Fanuc TP program (LS listing): OP5_LRG_SEQCHNG_AIR_D.LS

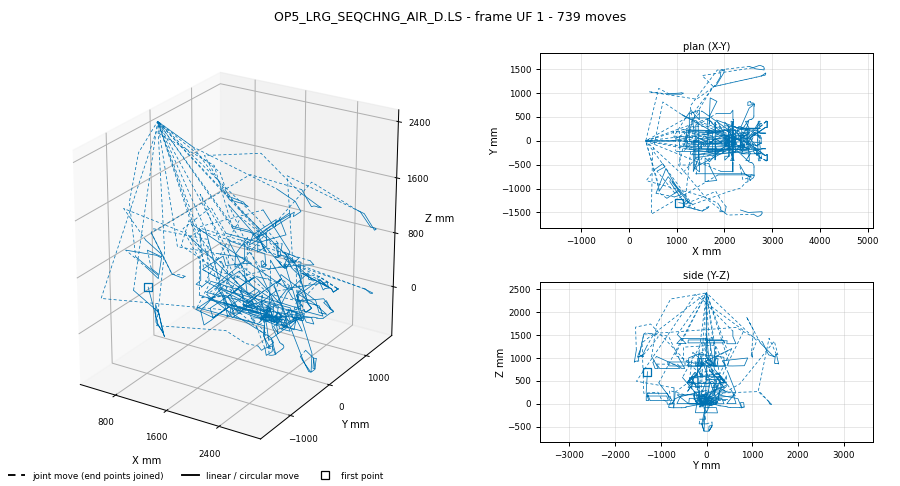
[picture p0: tool path of OP5_LRG_SEQCHNG_AIR_D.LS in frame UF 1, 739 of 740 moves have a stored position in this frame; points joined in program order, loops and branches not executed]
/PROG  OP5_LRG_SEQCHNG_AIR_D
/ATTR
OWNER		= MNEDITOR;
COMMENT		= "Large Main Base";
PROG_SIZE	= 95312;
CREATE		= DATE 26-02-26  TIME 11:37:22;
MODIFIED	= DATE 26-02-26  TIME 13:54:42;
FILE_NAME	= OP5_LRG_;
VERSION		= 0;
LINE_COUNT	= 2634;
MEMORY_SIZE	= 95996;
PROTECT		= READ_WRITE;
TCD:  STACK_SIZE	= 0,
      TASK_PRIORITY	= 50,
      TIME_SLICE	= 0,
      BUSY_LAMP_OFF	= 0,
      ABORT_REQUEST	= 0,
      PAUSE_REQUEST	= 0;
DEFAULT_GROUP	= 1,1,*,*,*;
CONTROL_CODE	= 00000000 00000000;
/APPL
  ARC Welding Equipment : 1,*,*,*,*;

MPAS ;
MPAS_NUM_PASSES        : 0;
MPAS_LAST_PASS         : 0;
MPAS_CURRENT_PASS      : 0;
MPAS_STATUS_PASS       : 0;
/MN
   1:  !********** WAR HAMMER ********** ;
   2:  !*------- FRAME LARGE ----------* ;
   3:  !*-- WELD SEQUENCE CHANGE 2026--* ;
   4:  !*------- FR500 CELL: D --------* ;
   5:  !******************************** ;
   6:   ;
   7:  CALL HOME    ;
   8:  UFRAME_NUM=1 ;
   9:  //DO[17:ON :SCAN ZONE2]=OFF ;
  10:   ;
  11:  !********POSITIONER MOVE******** ;
  12:J P[1] 85% CNT40    ;
  13:   ;
  14:L P[3] 1000mm/sec CNT40    ;
  15:   ;
  16:  !FR50L1000 ;
  17:  IF R[15:TECH HOLD]=1002,CALL TECH_HOLD ;
  18:   ;
  19:  !TO SKIP FRONT BUMPER WELDS ;
  20:  CALL ARC_DISABLE_FRONT_BMPR_LRG(0) ;
  21:   ;
  22:   ;
  23:   ;
  24:L P[5] 1000mm/sec FINE
    :  Arc Start[6]    ;
  25:  Weave Sine[6] ;
  26:  Track TAST[6] ;
  27:L P[6] WELD_SPEED FINE
    :  Arc End[6]    ;
  28:  Weave End ;
  29:  Track End ;
  30:   ;
  31:   ;
  32:   ;
  33:   ;
  34:L P[8] 800mm/sec CNT30    ;
  35:   ;
  36:L P[9] 1000mm/sec CNT30    ;
  37:   ;
  38:   ;
  39:  !FR50L1001 ;
  40:  IF R[15:TECH HOLD]=1003,CALL TECH_HOLD ;
  41:   ;
  42:   ;
  43:   ;
  44:   ;
  45:L P[10] 1000mm/sec FINE
    :  Arc Start[6]    ;
  46:  Weave Sine[6] ;
  47:  Track TAST[6] ;
  48:L P[11] WELD_SPEED FINE
    :  Arc End[6]    ;
  49:  Weave End ;
  50:  Track End ;
  51:   ;
  52:   ;
  53:   ;
  54:L P[12] 1000mm/sec CNT100    ;
  55:   ;
  56:   ;
  57:  !FR50L1002 ;
  58:  IF R[15:TECH HOLD]=1004,CALL TECH_HOLD ;
  59:   ;
  60:   ;
  61:L P[13] 1000mm/sec CNT70    ;
  62:   ;
  63:   ;
  64:   ;
  65:L P[14] 1000mm/sec FINE
    :  Arc Start[6]    ;
  66:  Weave Sine[6] ;
  67:  Track TAST[6] ;
  68:L P[15] WELD_SPEED FINE
    :  Arc End[6]    ;
  69:  Weave End ;
  70:  Track End ;
  71:   ;
  72:   ;
  73:   ;
  74:  CALL ARC_DISABLE_FRONT_BMPR_LRG(1) ;
  75:   ;
  76:L P[16] 1000mm/sec CNT100    ;
  77:   ;
  78:  !HOME ;
  79:J P[4] 70% CNT30    ;
  80:   ;
  81:  !********POSITIONER MOVE******** ;
  82:J P[17] 85% CNT30    ;
  83:   ;
  84:J P[18] 50% CNT100    ;
  85:   ;
  86:L P[19] 1000mm/sec CNT100    ;
  87:   ;
  88:   ;
  89:  !FR50L1003 ;
  90:  IF R[15:TECH HOLD]=1005,CALL TECH_HOLD ;
  91:   ;
  92:   ;
  93:L P[20] 1000mm/sec CNT25    ;
  94:   ;
  95:   ;
  96:   ;
  97:L P[21] 1000mm/sec FINE
    :  Arc Start[6]    ;
  98:  Weave Sine[6] ;
  99:  Track TAST[6] ;
 100:L P[22] WELD_SPEED CNT100    ;
 101:L P[23] WELD_SPEED FINE
    :  Arc End[6]    ;
 102:  Track End ;
 103:  Weave End ;
 104:   ;
 105:   ;
 106:   ;
 107:L P[24] 1000mm/sec CNT30    ;
 108:   ;
 109:   ;
 110:  !FR50L1010 ;
 111:  IF R[15:TECH HOLD]=1012,CALL TECH_HOLD ;
 112:   ;
 113:   ;
 114:L P[25] 1000mm/sec CNT30    ;
 115:   ;
 116:   ;
 117:   ;
 118:L P[26] 1000mm/sec FINE
    :  Arc Start[6]    ;
 119:  Weave Sine[6] ;
 120:  Track TAST[6] ;
 121:L P[27] WELD_SPEED CNT100    ;
 122:L P[28] WELD_SPEED FINE
    :  Arc End[6]    ;
 123:  Weave End ;
 124:  Track End ;
 125:   ;
 126:   ;
 127:   ;
 128:L P[29] 1000mm/sec CNT25    ;
 129:   ;
 130:   ;
 131:  !FR50L1020 ;
 132:  IF R[15:TECH HOLD]=1022,CALL TECH_HOLD ;
 133:   ;
 134:   ;
 135:J P[30] 50% CNT25    ;
 136:   ;
 137:   ;
 138:   ;
 139:L P[31] 1000mm/sec FINE
    :  Arc Start[6]    ;
 140:  Weave Sine[6] ;
 141:  Track TAST[6] ;
 142:L P[32] WELD_SPEED FINE
    :  Arc End[6]    ;
 143:  Weave End ;
 144:  Track End ;
 145:   ;
 146:   ;
 147:   ;
 148:L P[33] 1000mm/sec CNT30    ;
 149:   ;
 150:L P[34] 1000mm/sec CNT30    ;
 151:   ;
 152:   ;
 153:  !FR50L1030 ;
 154:  IF R[15:TECH HOLD]=1032,CALL TECH_HOLD ;
 155:   ;
 156:   ;
 157:   ;
 158:   ;
 159:L P[35] 1000mm/sec FINE
    :  Arc Start[6]    ;
 160:  Weave Sine[6] ;
 161:  Track TAST[6] ;
 162:L P[36] WELD_SPEED FINE
    :  Arc End[6]    ;
 163:  Weave End ;
 164:  Track End ;
 165:   ;
 166:   ;
 167:   ;
 168:L P[37] 1000mm/sec CNT50    ;
 169:   ;
 170:J P[38] 50% CNT50    ;
 171:   ;
 172:L P[39] 1000mm/sec CNT25    ;
 173:   ;
 174:   ;
 175:  !FR50L1040 ;
 176:  IF R[15:TECH HOLD]=1042,CALL TECH_HOLD ;
 177:   ;
 178:   ;
 179:   ;
 180:   ;
 181:L P[40] 1000mm/sec FINE
    :  Arc Start[6]    ;
 182:  Weave Sine[6] ;
 183:L P[41] WELD_SPEED FINE
    :  Arc End[6]    ;
 184:  Weave End ;
 185:   ;
 186:   ;
 187:   ;
 188:L P[42] 1000mm/sec CNT30    ;
 189:   ;
 190:L P[43] 1000mm/sec CNT70    ;
 191:   ;
 192:J P[44] 50% CNT50    ;
 193:   ;
 194:L P[45] 1000mm/sec CNT30    ;
 195:   ;
 196:   ;
 197:  !FR50L1050 ;
 198:  IF R[15:TECH HOLD]=1052,CALL TECH_HOLD ;
 199:   ;
 200:   ;
 201:   ;
 202:   ;
 203:L P[46] 1000mm/sec FINE
    :  Arc Start[6]    ;
 204:  Weave Sine[6] ;
 205:L P[47] WELD_SPEED FINE
    :  Arc End[6]    ;
 206:  Weave End ;
 207:   ;
 208:   ;
 209:   ;
 210:L P[48] 1000mm/sec CNT80    ;
 211:   ;
 212:J P[49] 50% CNT25    ;
 213:   ;
 214:L P[50] 1000mm/sec CNT25    ;
 215:   ;
 216:   ;
 217:  !FR50L1060 ;
 218:  IF R[15:TECH HOLD]=1062,CALL TECH_HOLD ;
 219:   ;
 220:   ;
 221:   ;
 222:   ;
 223:L P[51] 1000mm/sec FINE
    :  Arc Start[6]    ;
 224:  Weave Sine[6] ;
 225:L P[52] WELD_SPEED FINE
    :  Arc End[6]    ;
 226:  Weave End ;
 227:   ;
 228:   ;
 229:   ;
 230:L P[53] 500mm/sec CNT100    ;
 231:   ;
 232:L P[54] 1500mm/sec CNT35    ;
 233:   ;
 234:J P[55] 50% CNT30    ;
 235:   ;
 236:L P[56] 1000mm/sec CNT30    ;
 237:   ;
 238:   ;
 239:  !FR50L1070 ;
 240:  IF R[15:TECH HOLD]=1072,CALL TECH_HOLD ;
 241:   ;
 242:   ;
 243:   ;
 244:   ;
 245:L P[57] 1000mm/sec FINE
    :  Arc Start[6]    ;
 246:  Weave Sine[6] ;
 247:  Track TAST[6] ;
 248:L P[58] WELD_SPEED FINE
    :  Arc End[6]    ;
 249:  Weave End ;
 250:  Track End ;
 251:   ;
 252:   ;
 253:   ;
 254:L P[59] 1000mm/sec CNT100    ;
 255:   ;
 256:L P[60] 1000mm/sec CNT80    ;
 257:   ;
 258:   ;
 259:  !FR50L1080 ;
 260:  IF R[15:TECH HOLD]=1082,CALL TECH_HOLD ;
 261:   ;
 262:   ;
 263:   ;
 264:   ;
 265:L P[61] 1000mm/sec FINE
    :  Arc Start[6]    ;
 266:  Weave Sine[6] ;
 267:  Track TAST[6] ;
 268:L P[62] WELD_SPEED FINE
    :  Arc End[6]    ;
 269:  Weave End ;
 270:  Track End ;
 271:   ;
 272:   ;
 273:   ;
 274:J P[63] 30% CNT100    ;
 275:   ;
 276:J P[64] 50% CNT100    ;
 277:   ;
 278:L P[65] 1000mm/sec CNT80    ;
 279:   ;
 280:   ;
 281:  !FR50L1090 ;
 282:  IF R[15:TECH HOLD]=1092,CALL TECH_HOLD ;
 283:  !10MM PASS ;
 284:   ;
 285:   ;
 286:   ;
 287:   ;
 288:L P[66] 1000mm/sec FINE
    :  Arc Start[6]    ;
 289:  Weave Sine[6] ;
 290:  Track TAST[6] RPM[1] ;
 291:L P[67] WELD_SPEED CNT100    ;
 292:L P[68] WELD_SPEED CNT100    ;
 293:C P[69]
    :  P[70] WELD_SPEED CNT100    ;
 294:L P[71] WELD_SPEED FINE
    :  Arc End[6]    ;
 295:  Track End ;
 296:  Weave End ;
 297:   ;
 298:   ;
 299:   ;
 300:J P[72] 16% CNT25    ;
 301:   ;
 302:J P[74] 50% CNT25    ;
 303:   ;
 304:L P[75] 1000mm/sec CNT25    ;
 305:   ;
 306:   ;
 307:  !FR50L1100 ;
 308:  IF R[15:TECH HOLD]=1102,CALL TECH_HOLD ;
 309:   ;
 310:   ;
 311:   ;
 312:   ;
 313:L P[76] 1000mm/sec FINE
    :  Arc Start[6]    ;
 314:  Weave Sine[6] ;
 315:  Track TAST[6] RPM[2] ;
 316:L P[77] WELD_SPEED CNT100    ;
 317:L P[78] WELD_SPEED CNT100    ;
 318:C P[79]
    :  P[80] WELD_SPEED CNT100    ;
 319:L P[81] WELD_SPEED FINE
    :  Arc End[6]    ;
 320:  Weave End ;
 321:  Track End ;
 322:   ;
 323:   ;
 324:   ;
 325:J P[82] 50% CNT10    ;
 326:   ;
 327:J P[83] 50% CNT80    ;
 328:   ;
 329:L P[84] 1000mm/sec CNT25    ;
 330:   ;
 331:   ;
 332:  !FR50L1110MP1 ;
 333:  IF R[15:TECH HOLD]=1112,CALL TECH_HOLD ;
 334:   ;
 335:   ;
 336:  MP Offset  PR[3] RPM[1] ;
 337:   ;
 338:   ;
 339:L P[66] 1000mm/sec FINE
    :  Arc Start[6]    ;
 340:  Weave Sine[6] ;
 341:L P[67] WELD_SPEED CNT100    ;
 342:L P[68] WELD_SPEED CNT100    ;
 343:C P[69]
    :  P[70] WELD_SPEED CNT100    ;
 344:L P[71] WELD_SPEED FINE
    :  Arc End[6]    ;
 345:  Track End ;
 346:  Weave End ;
 347:   ;
 348:   ;
 349:  MP Offset End ;
 350:   ;
 351:J P[91] 40% CNT10    ;
 352:   ;
 353:J P[92] 50% CNT30    ;
 354:   ;
 355:L P[93] 1000mm/sec CNT25    ;
 356:   ;
 357:   ;
 358:  !FR50M1110MP2 ;
 359:   ;
 360:   ;
 361:  MP Offset  PR[4] RPM[1] ;
 362:   ;
 363:   ;
 364:L P[66] 1000mm/sec FINE
    :  Arc Start[6]    ;
 365:  Weave Sine[6] ;
 366:L P[67] WELD_SPEED CNT100    ;
 367:L P[68] WELD_SPEED CNT100    ;
 368:C P[69]
    :  P[70] WELD_SPEED CNT100    ;
 369:L P[71] WELD_SPEED FINE
    :  Arc End[6]    ;
 370:  Track End ;
 371:  Weave End ;
 372:   ;
 373:  MP Offset End ;
 374:   ;
 375:J P[100] 50% CNT25    ;
 376:   ;
 377:J P[102] 50% CNT25    ;
 378:   ;
 379:L P[103] 1000mm/sec CNT25    ;
 380:   ;
 381:   ;
 382:  !FR50L1120MP3 ;
 383:  IF R[15:TECH HOLD]=1122,CALL TECH_HOLD ;
 384:   ;
 385:   ;
 386:  MP Offset  PR[1] RPM[2] ;
 387:   ;
 388:   ;
 389:L P[76] 1000mm/sec FINE
    :  Arc Start[6]    ;
 390:  Weave Sine[6] ;
 391:L P[77] WELD_SPEED CNT100    ;
 392:L P[78] WELD_SPEED CNT100    ;
 393:C P[79]
    :  P[80] WELD_SPEED CNT100    ;
 394:L P[81] WELD_SPEED FINE
    :  Arc End[6]    ;
 395:  Weave End ;
 396:  Track End ;
 397:   ;
 398:   ;
 399:  MP Offset End ;
 400:   ;
 401:J P[110] 50% CNT25    ;
 402:   ;
 403:J P[111] 50% CNT25    ;
 404:   ;
 405:L P[112] 1000mm/sec CNT25    ;
 406:   ;
 407:   ;
 408:  !FR501130MP4 ;
 409:   ;
 410:   ;
 411:  MP Offset  PR[2] RPM[2] ;
 412:   ;
 413:L P[76] 1000mm/sec FINE
    :  Arc Start[6]    ;
 414:  Weave Sine[6] ;
 415:L P[77] WELD_SPEED CNT100    ;
 416:L P[78] WELD_SPEED CNT100    ;
 417:C P[79]
    :  P[80] WELD_SPEED CNT100    ;
 418:L P[81] WELD_SPEED FINE
    :  Arc End[6]    ;
 419:  Weave End ;
 420:  Track End ;
 421:   ;
 422:  MP Offset End ;
 423:   ;
 424:J P[119] 50% CNT25    ;
 425:   ;
 426:J P[121] 50% CNT25    ;
 427:   ;
 428:L P[122] 1000mm/sec CNT25    ;
 429:   ;
 430:   ;
 431:  !FR50L1140 ;
 432:  IF R[15:TECH HOLD]=1142,CALL TECH_HOLD ;
 433:   ;
 434:   ;
 435:   ;
 436:   ;
 437:L P[185] 1000mm/sec FINE
    :  Arc Start[8]    ;
 438:  Weave Sine[8] ;
 439:L P[186] WELD_SPEED CNT100    ;
 440:C P[187]
    :  P[188] WELD_SPEED FINE
    :  Arc End[8]    ;
 441:  Weave End ;
 442:   ;
 443:   ;
 444:   ;
 445:L P[127] 1000mm/sec CNT25    ;
 446:   ;
 447:J P[128] 50% CNT25    ;
 448:   ;
 449:   ;
 450:  !FR50L1141 ;
 451:  IF R[15:TECH HOLD]=1143,CALL TECH_HOLD ;
 452:   ;
 453:   ;
 454:   ;
 455:   ;
 456:L P[192] 1000mm/sec FINE
    :  Arc Start[8]    ;
 457:  Weave Sine[8] ;
 458:L P[193] WELD_SPEED CNT100    ;
 459:C P[194]
    :  P[197] WELD_SPEED FINE
    :  Arc End[8]    ;
 460:  Weave End ;
 461:   ;
 462:   ;
 463:   ;
 464:L P[133] 1000mm/sec CNT25    ;
 465:   ;
 466:L P[134] 1000mm/sec CNT25    ;
 467:   ;
 468:J P[135] 50% CNT25    ;
 469:   ;
 470:L P[136] 1000mm/sec CNT50    ;
 471:   ;
 472:   ;
 473:  !FR50L1150 ;
 474:  IF R[15:TECH HOLD]=1152,CALL TECH_HOLD ;
 475:   ;
 476:   ;
 477:   ;
 478:   ;
 479:L P[198] 1000mm/sec FINE
    :  Arc Start[6]    ;
 480:  Weave Sine[6] ;
 481:  Track TAST[6] ;
 482:L P[199] WELD_SPEED FINE
    :  Arc End[6]    ;
 483:  Weave End ;
 484:  Track End ;
 485:   ;
 486:   ;
 487:   ;
 488:L P[139] 1000mm/sec CNT100    ;
 489:   ;
 490:L P[140] 1000mm/sec CNT50    ;
 491:   ;
 492:   ;
 493:  !FR50L1160 ;
 494:  IF R[15:TECH HOLD]=1162,CALL TECH_HOLD ;
 495:   ;
 496:   ;
 497:   ;
 498:L P[203] 1000mm/sec FINE
    :  Arc Start[6]    ;
 499:  Weave Sine[6] ;
 500:  Track TAST[6] ;
 501:L P[204] WELD_SPEED FINE
    :  Arc End[6]    ;
 502:  Weave End ;
 503:  Track End ;
 504:   ;
 505:   ;
 506:   ;
 507:L P[143] 1000mm/sec CNT30    ;
 508:   ;
 509:  !********POSITIONER MOVE******** ;
 510:J P[144] 85% CNT30    ;
 511:   ;
 512:L P[145] 1000mm/sec CNT100    ;
 513:   ;
 514:   ;
 515:  !FR50L1170 ;
 516:  IF R[15:TECH HOLD]=1172,CALL TECH_HOLD ;
 517:   ;
 518:   ;
 519:   ;
 520:   ;
 521:L P[205] 1000mm/sec FINE
    :  Arc Start[6]    ;
 522:  Weave Sine[6] ;
 523:  Track TAST[6] ;
 524:L P[208] WELD_SPEED FINE
    :  Arc End[6]    ;
 525:  Weave End ;
 526:  Track End ;
 527:   ;
 528:   ;
 529:   ;
 530:L P[148] 1000mm/sec CNT100    ;
 531:   ;
 532:L P[149] 1500mm/sec CNT100    ;
 533:   ;
 534:   ;
 535:  !FR50L1180 ;
 536:  IF R[15:TECH HOLD]=1182,CALL TECH_HOLD ;
 537:   ;
 538:   ;
 539:   ;
 540:   ;
 541:L P[209] 1000mm/sec FINE
    :  Arc Start[6]    ;
 542:  Weave Sine[6] ;
 543:  Track TAST[6] ;
 544:L P[212] WELD_SPEED FINE
    :  Arc End[6]    ;
 545:  Weave End ;
 546:  Track End ;
 547:   ;
 548:   ;
 549:   ;
 550:L P[152] 1000mm/sec CNT100    ;
 551:   ;
 552:  !HOME ;
 553:J P[7] 100% CNT30    ;
 554:   ;
 555:  !********POSITIONER MOVE******** ;
 556:J P[153] 80% CNT30    ;
 557:   ;
 558:J P[154] 50% CNT100    ;
 559:   ;
 560:L P[155] 1000mm/sec CNT25    ;
 561:   ;
 562:   ;
 563:  !FR50L1210 ;
 564:  IF R[15:TECH HOLD]=1212,CALL TECH_HOLD ;
 565:   ;
 566:   ;
 567:   ;
 568:   ;
 569:L P[213] 1000mm/sec FINE
    :  Arc Start[6]    ;
 570:  Weave Sine[6] ;
 571:  Track TAST[6] ;
 572:L P[216] WELD_SPEED CNT100    ;
 573:L P[217] WELD_SPEED FINE
    :  Arc End[6]    ;
 574:  Weave End ;
 575:  Track End ;
 576:   ;
 577:   ;
 578:   ;
 579:L P[159] 1000mm/sec CNT25    ;
 580:   ;
 581:L P[160] 1000mm/sec CNT25    ;
 582:   ;
 583:   ;
 584:  !FR50L1220 ;
 585:  IF R[15:TECH HOLD]=1222,CALL TECH_HOLD ;
 586:   ;
 587:   ;
 588:   ;
 589:   ;
 590:L P[218] 1000mm/sec FINE
    :  Arc Start[6]    ;
 591:  Weave Sine[6] ;
 592:  Track TAST[6] ;
 593:L P[221] WELD_SPEED CNT100    ;
 594:L P[222] WELD_SPEED FINE
    :  Arc End[6]    ;
 595:  Weave End ;
 596:  Track End ;
 597:   ;
 598:   ;
 599:   ;
 600:L P[163] 1000mm/sec CNT80    ;
 601:   ;
 602:L P[164] 1200mm/sec CNT25    ;
 603:   ;
 604:   ;
 605:  !FR50L1230 ;
 606:  IF R[15:TECH HOLD]=1232,CALL TECH_HOLD ;
 607:   ;
 608:   ;
 609:   ;
 610:   ;
 611:L P[223] 1000mm/sec FINE
    :  Arc Start[6]    ;
 612:  Weave Sine[6] ;
 613:  Track TAST[6] ;
 614:L P[226] WELD_SPEED CNT100    ;
 615:L P[227] WELD_SPEED FINE
    :  Arc End[6]    ;
 616:  Weave End ;
 617:  Track End ;
 618:   ;
 619:   ;
 620:   ;
 621:L P[167] 1000mm/sec CNT25    ;
 622:   ;
 623:L P[168] 1000mm/sec CNT25    ;
 624:   ;
 625:   ;
 626:  !FR50L1240 ;
 627:  IF R[15:TECH HOLD]=1242,CALL TECH_HOLD ;
 628:   ;
 629:   ;
 630:   ;
 631:   ;
 632:L P[228] 1000mm/sec FINE
    :  Arc Start[6]    ;
 633:  Weave Sine[6] ;
 634:  Track TAST[6] ;
 635:L P[229] WELD_SPEED CNT100    ;
 636:L P[231] WELD_SPEED FINE
    :  Arc End[6]    ;
 637:  Weave End ;
 638:  Track End ;
 639:   ;
 640:   ;
 641:   ;
 642:L P[172] 1000mm/sec CNT25    ;
 643:   ;
 644:L P[173] 1000mm/sec CNT100    ;
 645:   ;
 646:  !HOME ;
 647:J P[116] 100% CNT100    ;
 648:   ;
 649:   ;
 650:  !********POSITIONER MOVE******** ;
 651:J P[174] 85% FINE    ;
 652:   ;
 653:  CALL T_CLEAN    ;
 654:   ;
 655:J P[175] 50% CNT35    ;
 656:   ;
 657:L P[176] 1000mm/sec CNT25    ;
 658:   ;
 659:   ;
 660:  !FR50L1250 ;
 661:  IF R[15:TECH HOLD]=1252,CALL TECH_HOLD ;
 662:   ;
 663:   ;
 664:   ;
 665:   ;
 666:L P[232] 1000mm/sec FINE
    :  Arc Start[6]    ;
 667:  Weave Sine[6] ;
 668:  Track TAST[6] ;
 669:L P[236] WELD_SPEED CNT100    ;
 670:L P[237] WELD_SPEED CNT100    ;
 671:L P[238] WELD_SPEED FINE
    :  Arc End[6]    ;
 672:  Weave End ;
 673:  Track End ;
 674:   ;
 675:   ;
 676:   ;
 677:L P[181] 1000mm/sec CNT100    ;
 678:   ;
 679:J P[182] 50% CNT100    ;
 680:   ;
 681:L P[184] 500mm/sec CNT100    ;
 682:   ;
 683:   ;
 684:  !FR50L1260 ;
 685:  IF R[15:TECH HOLD]=1262,CALL TECH_HOLD ;
 686:   ;
 687:   ;
 688:   ;
 689:   ;
 690:L P[239] 1000mm/sec FINE
    :  Arc Start[6]    ;
 691:  Weave Sine[6] ;
 692:  Track TAST[6] ;
 693:L P[244] WELD_SPEED CNT100    ;
 694:L P[245] WELD_SPEED CNT100    ;
 695:L P[246] WELD_SPEED FINE
    :  Arc End[6]    ;
 696:  Weave End ;
 697:  Track End ;
 698:   ;
 699:   ;
 700:   ;
 701:L P[189] 1000mm/sec CNT25    ;
 702:   ;
 703:J P[190] 50% CNT25    ;
 704:   ;
 705:L P[191] 1000mm/sec CNT25    ;
 706:   ;
 707:   ;
 708:  !FR50L1270 ;
 709:  IF R[15:TECH HOLD]=1272,CALL TECH_HOLD ;
 710:   ;
 711:   ;
 712:   ;
 713:   ;
 714:L P[247] 1000mm/sec FINE
    :  Arc Start[6]    ;
 715:  Weave Sine[6] ;
 716:  Track TAST[6] ;
 717:L P[250] WELD_SPEED CNT100    ;
 718:  Track End ;
 719:L P[251] WELD_SPEED FINE
    :  Arc End[6]    ;
 720:  Weave End ;
 721:  Track End ;
 722:   ;
 723:   ;
 724:   ;
 725:L P[195] 1000mm/sec CNT80    ;
 726:   ;
 727:L P[196] 1000mm/sec CNT100    ;
 728:   ;
 729:   ;
 730:  !FR50L1280 ;
 731:  IF R[15:TECH HOLD]=1282,CALL TECH_HOLD ;
 732:   ;
 733:   ;
 734:   ;
 735:   ;
 736:L P[253] 1000mm/sec FINE
    :  Arc Start[6]    ;
 737:  Weave Sine[6] ;
 738:  Track TAST[6] ;
 739:L P[254] WELD_SPEED CNT100    ;
 740:  Track End ;
 741:L P[255] WELD_SPEED FINE
    :  Arc End[6]    ;
 742:  Weave End ;
 743:  Track End ;
 744:   ;
 745:   ;
 746:   ;
 747:L P[200] 1000mm/sec CNT25    ;
 748:   ;
 749:J P[201] 50% CNT25    ;
 750:   ;
 751:L P[202] 1000mm/sec CNT25    ;
 752:   ;
 753:   ;
 754:  !FR50L1290 ;
 755:  IF R[15:TECH HOLD]=1292,CALL TECH_HOLD ;
 756:   ;
 757:   ;
 758:   ;
 759:   ;
 760:L P[257] 1000mm/sec FINE
    :  Arc Start[6]    ;
 761:  Weave Sine[6] ;
 762:  Track TAST[6] ;
 763:L P[258] WELD_SPEED CNT100    ;
 764:L P[259] WELD_SPEED FINE
    :  Arc End[6]    ;
 765:  Weave End ;
 766:  Track End ;
 767:L P[262] 1000mm/sec FINE
    :  Arc Start[6]    ;
 768:  Weave Sine[6] ;
 769:  Track TAST[6] ;
 770:L P[263] WELD_SPEED CNT100    ;
 771:L P[264] WELD_SPEED FINE
    :  Arc End[6]    ;
 772:  Weave End ;
 773:  Track End ;
 774:   ;
 775:   ;
 776:   ;
 777:L P[206] 1000mm/sec CNT100    ;
 778:   ;
 779:L P[207] 1000mm/sec CNT100    ;
 780:   ;
 781:   ;
 782:  !FR50L1300 ;
 783:  IF R[15:TECH HOLD]=1302,CALL TECH_HOLD ;
 784:   ;
 785:   ;
 786:   ;
 787:L P[90] 1000mm/sec FINE
    :  Arc Start[6]    ;
 788:  Weave Sine[6] ;
 789:  Track TAST[6] ;
 790:L P[98] WELD_SPEED CNT100    ;
 791:L P[101] WELD_SPEED FINE
    :  Arc End[6]    ;
 792:  Weave End ;
 793:  Track End ;
 794:   ;
 795:   ;
 796:L P[210] 1000mm/sec CNT100    ;
 797:   ;
 798:L P[211] 1000mm/sec CNT100    ;
 799:   ;
 800:   ;
 801:  !FR50L1310 ;
 802:  IF R[15:TECH HOLD]=1312,CALL TECH_HOLD ;
 803:   ;
 804:   ;
 805:   ;
 806:   ;
 807:L P[266] 1000mm/sec FINE
    :  Arc Start[6]    ;
 808:  Weave Sine[6] ;
 809:  Track TAST[6] ;
 810:L P[267] WELD_SPEED FINE
    :  Arc End[6]    ;
 811:  Weave End ;
 812:  Track End ;
 813:   ;
 814:   ;
 815:   ;
 816:L P[214] 1000mm/sec CNT100    ;
 817:   ;
 818:L P[215] 1000mm/sec CNT100    ;
 819:   ;
 820:   ;
 821:  !FR50L1320 ;
 822:  IF R[15:TECH HOLD]=1322,CALL TECH_HOLD ;
 823:   ;
 824:   ;
 825:   ;
 826:   ;
 827:L P[268] 1000mm/sec FINE
    :  Arc Start[6]    ;
 828:  Weave Sine[6] ;
 829:  Track TAST[6] ;
 830:L P[274] WELD_SPEED CNT100    ;
 831:L P[275] WELD_SPEED FINE
    :  Arc End[6]    ;
 832:  Weave End ;
 833:  Track End ;
 834:   ;
 835:   ;
 836:   ;
 837:L P[219] 1000mm/sec CNT100    ;
 838:   ;
 839:L P[220] 1000mm/sec CNT100    ;
 840:   ;
 841:J P[73] 50% CNT30    ;
 842:   ;
 843:  !********POSITIONER MOVE******** ;
 844:J P[86] 100% CNT30    ;
 845:   ;
 846:  !FR50L1330 ;
 847:  IF R[15:TECH HOLD]=1332,CALL TECH_HOLD ;
 848:   ;
 849:   ;
 850:J P[327] 40% CNT10    ;
 851:   ;
 852:   ;
 853:   ;
 854:L P[277] 1000mm/sec FINE
    :  Arc Start[8]    ;
 855:  Weave Sine[8] ;
 856:L P[278] WELD_SPEED FINE
    :  Arc End[8]    ;
 857:  Weave End ;
 858:   ;
 859:   ;
 860:   ;
 861:J P[85] 50% CNT30    ;
 862:   ;
 863:L P[233] 1000mm/sec CNT25    ;
 864:   ;
 865:  !********POSITIONER MOVE******** ;
 866:J P[225] 80% CNT20    ;
 867:   ;
 868:   ;
 869:   ;
 870:  !FR50L1340 ;
 871:  IF R[15:TECH HOLD]=1342,CALL TECH_HOLD ;
 872:   ;
 873:   ;
 874:   ;
 875:   ;
 876:L P[279] 1000mm/sec FINE
    :  Arc Start[6]    ;
 877:  Weave Sine[6] ;
 878:L P[282] WELD_SPEED FINE
    :  Arc End[6]    ;
 879:  Weave End ;
 880:   ;
 881:   ;
 882:   ;
 883:   ;
 884:  !FR50L1350 ;
 885:  IF R[15:TECH HOLD]=1352,CALL TECH_HOLD ;
 886:   ;
 887:   ;
 888:   ;
 889:   ;
 890:L P[283] 1000mm/sec FINE
    :  Arc Start[6]    ;
 891:  Weave Sine[6] ;
 892:L P[284] WELD_SPEED FINE
    :  Arc End[6]    ;
 893:  Weave End ;
 894:   ;
 895:   ;
 896:   ;
 897:L P[230] 1000mm/sec CNT25    ;
 898:   ;
 899:  !HOME ;
 900:J P[117] 100% CNT50    ;
 901:   ;
 902:  !********POSITIONER MOVE******** ;
 903:J P[768] 85% CNT25    ;
 904:   ;
 905:L P[234] 1000mm/sec CNT25    ;
 906:   ;
 907:J P[235] 50% CNT25    ;
 908:   ;
 909:   ;
 910:  !FR50L1380 ;
 911:  IF R[15:TECH HOLD]=1382,CALL TECH_HOLD ;
 912:   ;
 913:   ;
 914:   ;
 915:   ;
 916:L P[288] 1000mm/sec FINE
    :  Arc Start[6]    ;
 917:  Weave Sine[6] ;
 918:  Track TAST[6] ;
 919:L P[289] WELD_SPEED CNT100    ;
 920:L P[293] WELD_SPEED CNT100    ;
 921:L P[294] WELD_SPEED FINE
    :  Arc End[6]    ;
 922:  Weave End ;
 923:  Track End ;
 924:   ;
 925:   ;
 926:   ;
 927:L P[240] 800mm/sec CNT2    ;
 928:   ;
 929:L P[241] 800mm/sec CNT25    ;
 930:   ;
 931:  !********POSITIONER MOVE******** ;
 932:J P[242] 75% CNT5    ;
 933:   ;
 934:L P[243] 1000mm/sec CNT25    ;
 935:   ;
 936:   ;
 937:  !FR50L1390 ;
 938:  IF R[15:TECH HOLD]=1392,CALL TECH_HOLD ;
 939:   ;
 940:   ;
 941:   ;
 942:L P[297] 1000mm/sec FINE
    :  Arc Start[6]    ;
 943:  Weave Sine[6] ;
 944:L P[298] WELD_SPEED CNT100    ;
 945:L P[304] WELD_SPEED CNT100    ;
 946:L P[305] WELD_SPEED FINE
    :  Arc End[6]    ;
 947:  Weave End ;
 948:   ;
 949:   ;
 950:   ;
 951:L P[248] 1000mm/sec CNT25    ;
 952:   ;
 953:L P[249] 1000mm/sec CNT25    ;
 954:   ;
 955:   ;
 956:  !FR50L1400 ;
 957:  IF R[15:TECH HOLD]=1402,CALL TECH_HOLD ;
 958:   ;
 959:   ;
 960:   ;
 961:   ;
 962:L P[306] 1000mm/sec FINE
    :  Arc Start[6]    ;
 963:  Weave Sine[6] ;
 964:  Track TAST[6] ;
 965:L P[310] WELD_SPEED FINE
    :  Arc End[6]    ;
 966:  Weave End ;
 967:  Track End ;
 968:   ;
 969:   ;
 970:   ;
 971:L P[252] 1000mm/sec CNT25    ;
 972:   ;
 973:   ;
 974:  !FR50L1410 ;
 975:  IF R[15:TECH HOLD]=1412,CALL TECH_HOLD ;
 976:   ;
 977:   ;
 978:   ;
 979:   ;
 980:L P[311] 1000mm/sec FINE
    :  Arc Start[6]    ;
 981:  Weave Sine[6] ;
 982:  Track TAST[6] ;
 983:L P[312] WELD_SPEED CNT100    ;
 984:L P[313] WELD_SPEED FINE
    :  Arc End[6]    ;
 985:  Weave End ;
 986:  Track End ;
 987:   ;
 988:   ;
 989:   ;
 990:L P[256] 1000mm/sec CNT25    ;
 991:   ;
 992:   ;
 993:  !FR50L1420 ;
 994:  IF R[15:TECH HOLD]=1422,CALL TECH_HOLD ;
 995:   ;
 996:   ;
 997:   ;
 998:   ;
 999:L P[314] 1000mm/sec FINE
    :  Arc Start[6]    ;
1000:  Weave Sine[6] ;
1001:  Track TAST[6] ;
1002:L P[315] WELD_SPEED CNT100    ;
1003:L P[316] WELD_SPEED FINE
    :  Arc End[6]    ;
1004:  Weave End ;
1005:  Track End ;
1006:   ;
1007:   ;
1008:   ;
1009:L P[260] 1000mm/sec CNT25    ;
1010:   ;
1011:L P[261] 1000mm/sec CNT25    ;
1012:   ;
1013:   ;
1014:  !FR50L1430 ;
1015:  IF R[15:TECH HOLD]=1432,CALL TECH_HOLD ;
1016:   ;
1017:   ;
1018:   ;
1019:   ;
1020:L P[317] 1000mm/sec FINE
    :  Arc Start[6]    ;
1021:  Weave Sine[6] ;
1022:L P[318] WELD_SPEED CNT100    ;
1023:  Weave End ;
1024:L P[319] WELD_SPEED FINE
    :  Arc End[6]    ;
1025:   ;
1026:   ;
1027:   ;
1028:L P[265] 1000mm/sec CNT25    ;
1029:   ;
1030:   ;
1031:  !FR50L1431 ;
1032:  IF R[15:TECH HOLD]=1433,CALL TECH_HOLD ;
1033:   ;
1034:   ;
1035:   ;
1036:   ;
1037:L P[320] 1000mm/sec FINE
    :  Arc Start[6]    ;
1038:  Weave Sine[6] ;
1039:L P[330] WELD_SPEED CNT100    ;
1040:L P[333] WELD_SPEED FINE
    :  Arc End[6]    ;
1041:  Weave End ;
1042:   ;
1043:   ;
1044:   ;
1045:L P[269] 1000mm/sec CNT25    ;
1046:   ;
1047:L P[270] 1000mm/sec CNT25    ;
1048:   ;
1049:L P[271] 1000mm/sec CNT50 Wjnt    ;
1050:   ;
1051:J P[272] 50% CNT25    ;
1052:   ;
1053:L P[273] 1000mm/sec CNT25    ;
1054:   ;
1055:   ;
1056:  !FR50L1440 ;
1057:  IF R[15:TECH HOLD]=1442,CALL TECH_HOLD ;
1058:   ;
1059:   ;
1060:   ;
1061:   ;
1062:L P[334] 1000mm/sec FINE
    :  Arc Start[6]    ;
1063:  Weave Sine[6] ;
1064:  Track TAST[6] ;
1065:L P[338] WELD_SPEED FINE
    :  Arc End[6]    ;
1066:  Weave End ;
1067:  Track End ;
1068:   ;
1069:   ;
1070:   ;
1071:L P[276] 1000mm/sec CNT25    ;
1072:   ;
1073:   ;
1074:  !FR50L1450 ;
1075:  IF R[15:TECH HOLD]=1452,CALL TECH_HOLD ;
1076:   ;
1077:   ;
1078:   ;
1079:   ;
1080:L P[339] 1000mm/sec FINE
    :  Arc Start[6]    ;
1081:  Weave Sine[6] ;
1082:  Track TAST[6] ;
1083:L P[343] WELD_SPEED CNT100    ;
1084:L P[344] WELD_SPEED FINE
    :  Arc End[6]    ;
1085:  Weave End ;
1086:  Track End ;
1087:   ;
1088:   ;
1089:   ;
1090:L P[280] 1000mm/sec CNT25    ;
1091:   ;
1092:L P[281] 1000mm/sec CNT25    ;
1093:   ;
1094:   ;
1095:  !FR50L1460 ;
1096:  IF R[15:TECH HOLD]=1462,CALL TECH_HOLD ;
1097:   ;
1098:   ;
1099:   ;
1100:   ;
1101:L P[345] 1000mm/sec FINE
    :  Arc Start[6]    ;
1102:  Weave Sine[6] ;
1103:  Track TAST[6] ;
1104:L P[352] WELD_SPEED CNT100    ;
1105:L P[353] WELD_SPEED FINE
    :  Arc End[6]    ;
1106:  Weave End ;
1107:  Track End ;
1108:   ;
1109:   ;
1110:   ;
1111:L P[285] 1000mm/sec CNT25    ;
1112:   ;
1113:  !********POSITIONER MOVE******** ;
1114:J P[286] 75% CNT15    ;
1115:   ;
1116:L P[287] 1000mm/sec CNT25    ;
1117:   ;
1118:   ;
1119:  !FR50L1470 ;
1120:  IF R[15:TECH HOLD]=1472,CALL TECH_HOLD ;
1121:   ;
1122:   ;
1123:   ;
1124:   ;
1125:L P[354] 1000mm/sec FINE
    :  Arc Start[6]    ;
1126:  Weave Sine[6] ;
1127:  Track TAST[6] ;
1128:L P[355] WELD_SPEED FINE
    :  Arc End[6]    ;
1129:  Weave End ;
1130:  Track End ;
1131:   ;
1132:   ;
1133:   ;
1134:L P[290] 1000mm/sec CNT25    ;
1135:   ;
1136:  !********POSITIONER MOVE******** ;
1137:J P[291] 85% CNT2    ;
1138:   ;
1139:L P[292] 1000mm/sec CNT25    ;
1140:   ;
1141:   ;
1142:  !FR50L1480 ;
1143:  IF R[15:TECH HOLD]=1482,CALL TECH_HOLD ;
1144:   ;
1145:   ;
1146:   ;
1147:   ;
1148:L P[356] 1000mm/sec FINE
    :  Arc Start[8]    ;
1149:  Weave Sine[8] ;
1150:L P[357] WELD_SPEED FINE
    :  Arc End[8]    ;
1151:  Weave End ;
1152:   ;
1153:   ;
1154:   ;
1155:L P[295] 1000mm/sec CNT25    ;
1156:   ;
1157:L P[296] 1000mm/sec CNT25    ;
1158:   ;
1159:   ;
1160:  !FR50L1490 ;
1161:  IF R[15:TECH HOLD]=1492,CALL TECH_HOLD ;
1162:   ;
1163:   ;
1164:   ;
1165:   ;
1166:L P[358] 1000mm/sec FINE
    :  Arc Start[6]    ;
1167:  Weave Sine[6] ;
1168:  Track TAST[6] ;
1169:L P[359] WELD_SPEED FINE
    :  Arc End[6]    ;
1170:  Weave End ;
1171:  Track End ;
1172:   ;
1173:   ;
1174:   ;
1175:L P[299] 1000mm/sec CNT25    ;
1176:   ;
1177:L P[300] 1000mm/sec CNT25    ;
1178:   ;
1179:L P[301] 1000mm/sec CNT25    ;
1180:   ;
1181:  !********POSITIONER MOVE******** ;
1182:J P[302] 85% FINE    ;
1183:   ;
1184:L P[303] 1000mm/sec CNT25    ;
1185:   ;
1186:   ;
1187:  !FR50L1500 ;
1188:  IF R[15:TECH HOLD]=1502,CALL TECH_HOLD ;
1189:   ;
1190:   ;
1191:   ;
1192:   ;
1193:L P[362] 1000mm/sec FINE
    :  Arc Start[6]    ;
1194:  Weave Sine[6] ;
1195:L P[363] WELD_SPEED CNT100    ;
1196:L P[364] WELD_SPEED FINE
    :  Arc End[6]    ;
1197:  Weave End ;
1198:   ;
1199:   ;
1200:   ;
1201:L P[307] 1000mm/sec CNT25    ;
1202:   ;
1203:J P[308] 50% CNT25    ;
1204:   ;
1205:L P[309] 1000mm/sec CNT25    ;
1206:   ;
1207:   ;
1208:  !FR50L1510 ;
1209:  IF R[15:TECH HOLD]=1512,CALL TECH_HOLD ;
1210:   ;
1211:   ;
1212:   ;
1213:   ;
1214:L P[366] 1000mm/sec FINE
    :  Arc Start[6]    ;
1215:  Weave Sine[6] ;
1216:  Track TAST[6] ;
1217:L P[369] WELD_SPEED CNT100    ;
1218:C P[370]
    :  P[374] WELD_SPEED CNT100    ;
1219:L P[375] WELD_SPEED CNT100    ;
1220:C P[382]
    :  P[383] WELD_SPEED CNT100    ;
1221:L P[384] WELD_SPEED CNT100    ;
1222:C P[385]
    :  P[386] WELD_SPEED CNT100    ;
1223:L P[387] WELD_SPEED FINE
    :  Arc End[6]    ;
1224:  Weave End ;
1225:  Track End ;
1226:   ;
1227:   ;
1228:L P[321] 1000mm/sec CNT80    ;
1229:   ;
1230:J P[322] 40% CNT80    ;
1231:   ;
1232:  --eg:Insert g2j2 @90 Loadstop!!! ;
1233:   ;
1234:  !********POSITIONER MOVE******** ;
1235:J P[114] 85% CNT40    ;
1236:   ;
1237:J P[115] 50% CNT25    ;
1238:   ;
1239:  CALL ARC_DISABLE_RH_LS(0) ;
1240:   ;
1241:   ;
1242:  !FR50L2040 ;
1243:  IF R[15:TECH HOLD]=2042,CALL TECH_HOLD ;
1244:   ;
1245:   ;
1246:L P[473] 1000mm/sec CNT25    ;
1247:   ;
1248:   ;
1249:   ;
1250:L P[770] 1000mm/sec FINE
    :  Arc Start[8]    ;
1251:  Weave Sine[8] ;
1252:L P[771] WELD_SPEED CNT100    ;
1253:C P[772]
    :  P[773] WELD_SPEED CNT100    ;
1254:L P[774] WELD_SPEED CNT100    ;
1255:L P[775] WELD_SPEED CNT100    ;
1256:L P[776] WELD_SPEED CNT100    ;
1257:L P[777] WELD_SPEED FINE
    :  Arc End[8]    ;
1258:  Weave End ;
1259:   ;
1260:  CALL ARC_DISABLE_RH_LS(1) ;
1261:   ;
1262:L P[494] 1000mm/sec CNT25    ;
1263:   ;
1264:J P[497] 50% CNT75    ;
1265:   ;
1266:  --eg:Insert g2j2 @90 Loadstop!!! ;
1267:   ;
1268:   ;
1269:   ;
1270:  !********POSITIONER MOVE******** ;
1271:J P[502] 40% CNT40    ;
1272:   ;
1273:J P[323] 40% CNT25    ;
1274:   ;
1275:  !CELL ID: D - ;
1276:   ;
1277:L P[390] 1000mm/sec FINE
    :  Arc Start[1]    ;
1278:L P[391] WELD_SPEED FINE
    :  Arc End[1]    ;
1279:   ;
1280:J P[324] 50% CNT30    ;
1281:   ;
1282:L P[328] 800mm/sec CNT60    ;
1283:   ;
1284:J P[224] 40% CNT100    ;
1285:   ;
1286:J P[329] 40% CNT90    ;
1287:   ;
1288:J P[331] 50% CNT50    ;
1289:   ;
1290:L P[332] 1000mm/sec CNT25    ;
1291:   ;
1292:   ;
1293:  !FR50L1520 ;
1294:  IF R[15:TECH HOLD]=1522,CALL TECH_HOLD ;
1295:   ;
1296:   ;
1297:   ;
1298:   ;
1299:L P[399] 1000mm/sec FINE
    :  Arc Start[6]    ;
1300:  Weave Sine[6] ;
1301:  Track TAST[6] ;
1302:L P[400] WELD_SPEED FINE
    :  Arc End[6]    ;
1303:  Weave End ;
1304:  Track End ;
1305:   ;
1306:   ;
1307:   ;
1308:L P[335] 1000mm/sec CNT25    ;
1309:   ;
1310:J P[336] 50% CNT25    ;
1311:   ;
1312:L P[337] 1000mm/sec CNT25    ;
1313:   ;
1314:   ;
1315:  !FR50L1530 ;
1316:  IF R[15:TECH HOLD]=1532,CALL TECH_HOLD ;
1317:   ;
1318:   ;
1319:   ;
1320:   ;
1321:L P[401] 1000mm/sec FINE
    :  Arc Start[6]    ;
1322:  Weave Sine[6] ;
1323:  Track TAST[6] ;
1324:L P[402] WELD_SPEED FINE
    :  Arc End[6]    ;
1325:  Weave End ;
1326:  Track End ;
1327:   ;
1328:   ;
1329:   ;
1330:L P[340] 1000mm/sec CNT25    ;
1331:   ;
1332:L P[341] 1000mm/sec CNT25    ;
1333:   ;
1334:L P[342] 1000mm/sec CNT25    ;
1335:   ;
1336:  !FR50L1540 ;
1337:  IF R[15:TECH HOLD]=1542,CALL TECH_HOLD ;
1338:   ;
1339:   ;
1340:   ;
1341:L P[403] 1000mm/sec FINE
    :  Arc Start[6]    ;
1342:  Weave Sine[6] ;
1343:  Track TAST[6] ;
1344:L P[404] WELD_SPEED CNT100    ;
1345:L P[405] WELD_SPEED FINE
    :  Arc End[6]    ;
1346:  Weave End ;
1347:  Track End ;
1348:   ;
1349:   ;
1350:L P[346] 1000mm/sec CNT40    ;
1351:   ;
1352:L P[347] 1100mm/sec CNT50 Wjnt    ;
1353:   ;
1354:J P[348] 50% CNT35    ;
1355:   ;
1356:  --eg:Insert g2j2 @90 content ;
1357:   ;
1358:J P[88] 50% CNT90    ;
1359:   ;
1360:L P[96] 1000mm/sec CNT25    ;
1361:   ;
1362:   ;
1363:  !FR50L1590 ;
1364:  IF R[15:TECH HOLD]=1592,CALL TECH_HOLD ;
1365:   ;
1366:   ;
1367:   ;
1368:   ;
1369:L P[439] 1000mm/sec FINE
    :  Arc Start[6]    ;
1370:  Weave Sine[6] ;
1371:  Track TAST[6] ;
1372:L P[440] WELD_SPEED FINE
    :  Arc End[6]    ;
1373:  Weave End ;
1374:  Track End ;
1375:   ;
1376:   ;
1377:   ;
1378:L P[120] 1000mm/sec CNT25    ;
1379:   ;
1380:J P[123] 50% CNT25    ;
1381:   ;
1382:   ;
1383:  !FR50L1600 ;
1384:  IF R[15:TECH HOLD]=1602,CALL TECH_HOLD ;
1385:   ;
1386:   ;
1387:   ;
1388:   ;
1389:L P[441] 1000mm/sec FINE
    :  Arc Start[6]    ;
1390:  Weave Sine[6] ;
1391:  Track TAST[6] ;
1392:L P[442] WELD_SPEED FINE
    :  Arc End[6]    ;
1393:  Weave End ;
1394:  Track End ;
1395:   ;
1396:   ;
1397:   ;
1398:L P[126] 1000mm/sec CNT25    ;
1399:   ;
1400:J P[129] 50% CNT25    ;
1401:   ;
1402:   ;
1403:  !FR50L1601 ;
1404:  IF R[15:TECH HOLD]=1603,CALL TECH_HOLD ;
1405:   ;
1406:   ;
1407:   ;
1408:   ;
1409:L P[443] 1000mm/sec FINE
    :  Arc Start[6]    ;
1410:  Weave Sine[6] ;
1411:  Track TAST[6] ;
1412:L P[444] WELD_SPEED FINE
    :  Arc End[6]    ;
1413:  Weave End ;
1414:  Track End ;
1415:   ;
1416:   ;
1417:   ;
1418:L P[132] 1000mm/sec CNT25    ;
1419:   ;
1420:L P[137] 1200mm/sec CNT40 Wjnt    ;
1421:   ;
1422:  !********POSITIONER MOVE******** ;
1423:J P[138] 90% CNT30    ;
1424:   ;
1425:L P[141] 1000mm/sec CNT25    ;
1426:   ;
1427:L P[142] 1000mm/sec CNT25    ;
1428:   ;
1429:   ;
1430:  !FR50L1610 ;
1431:  IF R[15:TECH HOLD]=1612,CALL TECH_HOLD ;
1432:   ;
1433:   ;
1434:   ;
1435:   ;
1436:L P[445] 1000mm/sec FINE
    :  Arc Start[6]    ;
1437:  Weave Sine[6] ;
1438:  Track TAST[6] ;
1439:L P[446] WELD_SPEED CNT100    ;
1440:L P[447] WELD_SPEED FINE
    :  Arc End[6]    ;
1441:  Weave End ;
1442:  Track End ;
1443:   ;
1444:   ;
1445:   ;
1446:L P[151] 1000mm/sec CNT25    ;
1447:   ;
1448:L P[156] 1000mm/sec CNT25    ;
1449:   ;
1450:   ;
1451:   ;
1452:  !FR50L1620 ;
1453:  IF R[15:TECH HOLD]=1622,CALL TECH_HOLD ;
1454:   ;
1455:   ;
1456:   ;
1457:   ;
1458:L P[448] 1000mm/sec FINE
    :  Arc Start[6]    ;
1459:  Weave Sine[6] ;
1460:  Track TAST[6] ;
1461:L P[449] WELD_SPEED CNT100    ;
1462:L P[450] WELD_SPEED FINE
    :  Arc End[6]    ;
1463:  Weave End ;
1464:  Track End ;
1465:   ;
1466:   ;
1467:   ;
1468:L P[365] 1000mm/sec CNT75    ;
1469:   ;
1470:L P[376] 1000mm/sec CNT25    ;
1471:   ;
1472:J P[380] 50% CNT40    ;
1473:   ;
1474:  !********POSITIONER MOVE******** ;
1475:J P[504] 85% CNT30    ;
1476:   ;
1477:  CALL HOME    ;
1478:  CALL T_CLEAN    ;
1479:   ;
1480:J P[381] 90% CNT30    ;
1481:   ;
1482:J P[397] 50% CNT25    ;
1483:   ;
1484:   ;
1485:  !FR50L1630 ;
1486:  IF R[15:TECH HOLD]=1632,CALL TECH_HOLD ;
1487:   ;
1488:   ;
1489:   ;
1490:   ;
1491:L P[453] 1000mm/sec FINE
    :  Arc Start[6]    ;
1492:  Weave Sine[6] ;
1493:  Track TAST[6] ;
1494:L P[454] WELD_SPEED CNT100    ;
1495:C P[455]
    :  P[456] WELD_SPEED CNT100    ;
1496:L P[457] WELD_SPEED CNT100    ;
1497:C P[458]
    :  P[462] WELD_SPEED CNT100    ;
1498:L P[463] WELD_SPEED FINE
    :  Arc End[6]    ;
1499:  Weave End ;
1500:  Track End ;
1501:   ;
1502:   ;
1503:   ;
1504:L P[412] 1000mm/sec CNT40    ;
1505:   ;
1506:J P[413] 50% CNT35    ;
1507:   ;
1508:   ;
1509:  !FR50L1640 ;
1510:  IF R[15:TECH HOLD]=1642,CALL TECH_HOLD ;
1511:   ;
1512:   ;
1513:   ;
1514:   ;
1515:L P[464] 1000mm/sec FINE
    :  Arc Start[6]    ;
1516:  Weave Sine[6] ;
1517:  Track TAST[6] ;
1518:L P[465] WELD_SPEED CNT100    ;
1519:C P[466]
    :  P[467] WELD_SPEED CNT100    ;
1520:L P[468] WELD_SPEED CNT100    ;
1521:L P[474] WELD_SPEED CNT100    ;
1522:L P[475] WELD_SPEED CNT100    ;
1523:L P[476] WELD_SPEED CNT100    ;
1524:L P[481] WELD_SPEED FINE
    :  Arc End[6]    ;
1525:  Weave End ;
1526:  Track End ;
1527:   ;
1528:   ;
1529:   ;
1530:L P[432] 1000mm/sec CNT100    ;
1531:   ;
1532:J P[433] 50% CNT35    ;
1533:   ;
1534:  !********POSITIONER MOVE******** ;
1535:J P[434] 85% CNT30    ;
1536:   ;
1537:L P[435] 1000mm/sec CNT25    ;
1538:   ;
1539:J P[436] 50% CNT25    ;
1540:   ;
1541:   ;
1542:  !FR50L1650 ;
1543:  IF R[15:TECH HOLD]=1652,CALL TECH_HOLD ;
1544:   ;
1545:   ;
1546:   ;
1547:   ;
1548:L P[482] 1000mm/sec FINE
    :  Arc Start[6]    ;
1549:  Weave Sine[6] ;
1550:L P[486] WELD_SPEED CNT100    ;
1551:L P[487] WELD_SPEED CNT100    ;
1552:L P[493] WELD_SPEED CNT100    ;
1553:  Track TAST[6] ;
1554:L P[509] WELD_SPEED CNT100    ;
1555:L P[510] WELD_SPEED CNT100    ;
1556:L P[511] WELD_SPEED CNT100    ;
1557:L P[512] WELD_SPEED CNT100    ;
1558:C P[513]
    :  P[514] WELD_SPEED CNT100    ;
1559:L P[515] WELD_SPEED CNT100    ;
1560:C P[516]
    :  P[517] WELD_SPEED CNT100    ;
1561:L P[518] WELD_SPEED FINE
    :  Arc End[6]    ;
1562:  Weave End ;
1563:  Track End ;
1564:   ;
1565:   ;
1566:   ;
1567:L P[451] 1000mm/sec CNT100    ;
1568:   ;
1569:L P[452] 1000mm/sec CNT80    ;
1570:   ;
1571:   ;
1572:  !FR50L1651 ;
1573:  IF R[15:TECH HOLD]=1653,CALL TECH_HOLD ;
1574:   ;
1575:   ;
1576:   ;
1577:   ;
1578:L P[522] 1000mm/sec FINE
    :  Arc Start[6]    ;
1579:  Weave Sine[6] ;
1580:  Track TAST[6] ;
1581:L P[523] WELD_SPEED CNT100    ;
1582:C P[524]
    :  P[530] WELD_SPEED CNT100    ;
1583:C P[531]
    :  P[532] WELD_SPEED FINE
    :  Arc End[6]    ;
1584:  Weave End ;
1585:  Track End ;
1586:   ;
1587:   ;
1588:   ;
1589:L P[459] 1000mm/sec CNT60    ;
1590:   ;
1591:L P[460] 1000mm/sec CNT100    ;
1592:   ;
1593:J P[461] 50% CNT40    ;
1594:   ;
1595:J P[498] 50% CNT40    ;
1596:  --eg:Insert g2j2 @90 content ;
1597:   ;
1598:  !********POSITIONER MOVE******** ;
1599:J P[350] 90% CNT40    ;
1600:   ;
1601:J P[349] 50% CNT25    ;
1602:   ;
1603:L P[351] 1000mm/sec CNT25    ;
1604:   ;
1605:   ;
1606:  !FR50L1540 ;
1607:  IF R[15:TECH HOLD]=1542,CALL TECH_HOLD ;
1608:   ;
1609:   ;
1610:   ;
1611:   ;
1612:L P[778] 1000mm/sec FINE
    :  Arc Start[6]    ;
1613:  Weave Sine[6] ;
1614:  Track TAST[6] ;
1615:L P[779] WELD_SPEED CNT100    ;
1616:L P[780] WELD_SPEED CNT100    ;
1617:L P[781] WELD_SPEED CNT100    ;
1618:L P[782] WELD_SPEED CNT100    ;
1619:L P[783] WELD_SPEED CNT100    ;
1620:L P[784] WELD_SPEED CNT100    ;
1621:L P[785] WELD_SPEED FINE
    :  Arc End[6]    ;
1622:  Weave End ;
1623:  Track End ;
1624:   ;
1625:   ;
1626:   ;
1627:L P[360] 1000mm/sec CNT60    ;
1628:   ;
1629:L P[361] 1000mm/sec CNT25    ;
1630:   ;
1631:   ;
1632:  !FR50L1550 ;
1633:  IF R[15:TECH HOLD]=1552,CALL TECH_HOLD ;
1634:   ;
1635:   ;
1636:   ;
1637:   ;
1638:L P[416] 1000mm/sec FINE
    :  Arc Start[6]    ;
1639:  Weave Sine[6] ;
1640:  Track TAST[6] ;
1641:L P[417] WELD_SPEED CNT100    ;
1642:L P[418] WELD_SPEED CNT100    ;
1643:L P[419] WELD_SPEED CNT100    ;
1644:L P[420] WELD_SPEED FINE
    :  Arc End[6]    ;
1645:  Weave End ;
1646:  Track End ;
1647:   ;
1648:   ;
1649:   ;
1650:L P[367] 1000mm/sec CNT25    ;
1651:   ;
1652:L P[368] 1000mm/sec CNT40    ;
1653:   ;
1654:J P[183] 50% CNT40    ;
1655:   ;
1656:  !********POSITIONER MOVE******** ;
1657:J P[377] 90% CNT30    ;
1658:   ;
1659:J P[378] 50% CNT40    ;
1660:   ;
1661:J P[379] 50% CNT40    ;
1662:   ;
1663:   ;
1664:  !FR50L1570 ;
1665:  IF R[15:TECH HOLD]=1572,CALL TECH_HOLD ;
1666:   ;
1667:   ;
1668:   ;
1669:   ;
1670:L P[421] 1000mm/sec FINE
    :  Arc Start[6]    ;
1671:  Weave Sine[6] ;
1672:  Track TAST[6] ;
1673:L P[422] WELD_SPEED CNT100    ;
1674:L P[423] WELD_SPEED CNT100    ;
1675:L P[424] WELD_SPEED CNT100    ;
1676:L P[425] WELD_SPEED CNT100    ;
1677:L P[426] WELD_SPEED CNT100    ;
1678:L P[427] WELD_SPEED CNT100    ;
1679:L P[428] WELD_SPEED FINE
    :  Arc End[6]    ;
1680:  Weave End ;
1681:  Track End ;
1682:   ;
1683:   ;
1684:   ;
1685:L P[388] 1000mm/sec CNT100    ;
1686:   ;
1687:L P[389] 1000mm/sec CNT25    ;
1688:   ;
1689:   ;
1690:  !FR50L1580 ;
1691:  IF R[15:TECH HOLD]=1582,CALL TECH_HOLD ;
1692:   ;
1693:   ;
1694:   ;
1695:   ;
1696:L P[429] 1000mm/sec FINE
    :  Arc Start[6]    ;
1697:  Weave Sine[6] ;
1698:  Track TAST[6] ;
1699:L P[430] WELD_SPEED CNT100    ;
1700:L P[431] WELD_SPEED CNT100    ;
1701:L P[437] WELD_SPEED CNT100    ;
1702:L P[438] WELD_SPEED FINE
    :  Arc End[6]    ;
1703:  Weave End ;
1704:  Track End ;
1705:   ;
1706:   ;
1707:   ;
1708:L P[395] 600mm/sec CNT25    ;
1709:   ;
1710:L P[396] 1000mm/sec CNT100    ;
1711:   ;
1712:J P[326] 60% CNT25    ;
1713:   ;
1714:J P[325] 70% CNT30    ;
1715:   ;
1716:  !********POSITIONER MOVE******** ;
1717:J P[503] 90% CNT30    ;
1718:   ;
1719:J P[477] 50% CNT40    ;
1720:   ;
1721:J P[478] 50% CNT80    ;
1722:   ;
1723:J P[479] 50% CNT60    ;
1724:   ;
1725:J P[480] 50% CNT30    ;
1726:   ;
1727:   ;
1728:  !FR50L1660 ;
1729:  IF R[15:TECH HOLD]=1662,CALL TECH_HOLD ;
1730:   ;
1731:   ;
1732:   ;
1733:   ;
1734:L P[533] 1000mm/sec FINE
    :  Arc Start[6]    ;
1735:  Weave Sine[6] ;
1736:  Track TAST[6] ;
1737:L P[538] WELD_SPEED FINE
    :  Arc End[6]    ;
1738:  Weave End ;
1739:  Track End ;
1740:   ;
1741:   ;
1742:   ;
1743:J P[483] 20% CNT100    ;
1744:   ;
1745:J P[484] 60% CNT25    ;
1746:   ;
1747:L P[485] 600mm/sec CNT25    ;
1748:   ;
1749:   ;
1750:  !FR50L1661 ;
1751:  IF R[15:TECH HOLD]=1663,CALL TECH_HOLD ;
1752:   ;
1753:   ;
1754:   ;
1755:   ;
1756:L P[539] 1000mm/sec FINE
    :  Arc Start[6]    ;
1757:  Weave Sine[6] ;
1758:  Track TAST[6] ;
1759:L P[540] WELD_SPEED FINE
    :  Arc End[6]    ;
1760:  Weave End ;
1761:  Track End ;
1762:   ;
1763:   ;
1764:   ;
1765:L P[488] 500mm/sec CNT25    ;
1766:   ;
1767:L P[489] 500mm/sec CNT35    ;
1768:   ;
1769:L P[490] 1000mm/sec CNT25    ;
1770:   ;
1771:  !********POSITIONER MOVE******** ;
1772:J P[491] 90% CNT25    ;
1773:   ;
1774:L P[492] 1000mm/sec CNT25    ;
1775:   ;
1776:   ;
1777:  !FR50L1670 ;
1778:  IF R[15:TECH HOLD]=1672,CALL TECH_HOLD ;
1779:   ;
1780:   ;
1781:   ;
1782:   ;
1783:L P[541] 1000mm/sec FINE
    :  Arc Start[8]    ;
1784:  Weave Sine[8] ;
1785:L P[545] WELD_SPEED FINE
    :  Arc End[8]    ;
1786:  Weave End ;
1787:   ;
1788:   ;
1789:   ;
1790:L P[495] 800mm/sec CNT25    ;
1791:   ;
1792:L P[496] 1000mm/sec CNT25    ;
1793:   ;
1794:   ;
1795:  !FR50L1680 ;
1796:  IF R[15:TECH HOLD]=1682,CALL TECH_HOLD ;
1797:   ;
1798:   ;
1799:   ;
1800:   ;
1801:L P[546] 1000mm/sec FINE
    :  Arc Start[6]    ;
1802:  Weave Sine[6] ;
1803:  Track TAST[6] ;
1804:L P[550] WELD_SPEED FINE
    :  Arc End[6]    ;
1805:  Weave End ;
1806:  Track End ;
1807:   ;
1808:   ;
1809:   ;
1810:L P[499] 1000mm/sec CNT25    ;
1811:   ;
1812:  !********POSITIONER MOVE******** ;
1813:J P[500] 75% CNT20    ;
1814:   ;
1815:L P[501] 1000mm/sec CNT25    ;
1816:   ;
1817:   ;
1818:  !FR50L1690 ;
1819:  IF R[15:TECH HOLD]=1692,CALL TECH_HOLD ;
1820:   ;
1821:   ;
1822:   ;
1823:   ;
1824:L P[551] 1000mm/sec FINE
    :  Arc Start[6]    ;
1825:  Weave Sine[6] ;
1826:  Track TAST[6] ;
1827:L P[552] WELD_SPEED CNT100    ;
1828:L P[557] WELD_SPEED FINE
    :  Arc End[6]    ;
1829:  Weave End ;
1830:  Track End ;
1831:   ;
1832:   ;
1833:   ;
1834:L P[505] 300mm/sec CNT40    ;
1835:   ;
1836:L P[506] 1000mm/sec CNT40    ;
1837:   ;
1838:L P[507] 1000mm/sec CNT40    ;
1839:   ;
1840:   ;
1841:  !FR50L1700 ;
1842:  IF R[15:TECH HOLD]=1702,CALL TECH_HOLD ;
1843:   ;
1844:   ;
1845:   ;
1846:   ;
1847:L P[558] 1000mm/sec FINE
    :  Arc Start[6]    ;
1848:  Weave Sine[6] ;
1849:  Track TAST[6] ;
1850:L P[561] WELD_SPEED CNT100    ;
1851:C P[562]
    :  P[566] WELD_SPEED CNT100    ;
1852:L P[567] WELD_SPEED CNT100    ;
1853:C P[570]
    :  P[574] WELD_SPEED CNT100    ;
1854:L P[575] WELD_SPEED CNT100    ;
1855:C P[579]
    :  P[580] WELD_SPEED CNT100    ;
1856:L P[582] WELD_SPEED FINE
    :  Arc End[6]    ;
1857:  Weave End ;
1858:  Track End ;
1859:   ;
1860:   ;
1861:   ;
1862:L P[519] 1000mm/sec CNT100    ;
1863:   ;
1864:L P[520] 1000mm/sec CNT40    ;
1865:   ;
1866:L P[521] 500mm/sec CNT30    ;
1867:   ;
1868:   ;
1869:  !FR50L1710 ;
1870:  IF R[15:TECH HOLD]=1712,CALL TECH_HOLD ;
1871:   ;
1872:   ;
1873:   ;
1874:   ;
1875:L P[583] 1000mm/sec FINE
    :  Arc Start[6]    ;
1876:  Weave Sine[6] ;
1877:  Track TAST[6] ;
1878:L P[584] WELD_SPEED CNT100    ;
1879:L P[586] WELD_SPEED FINE
    :  Arc End[6]    ;
1880:  Weave End ;
1881:  Track End ;
1882:   ;
1883:   ;
1884:   ;
1885:L P[525] 500mm/sec CNT25    ;
1886:   ;
1887:L P[526] 800mm/sec CNT50 Wjnt    ;
1888:   ;
1889:L P[527] 1400mm/sec CNT100 Wjnt    ;
1890:   ;
1891:J P[528] 50% CNT100    ;
1892:   ;
1893:L P[529] 1000mm/sec CNT25    ;
1894:   ;
1895:   ;
1896:  !FR50L1720 ;
1897:  IF R[15:TECH HOLD]=1722,CALL TECH_HOLD ;
1898:   ;
1899:   ;
1900:   ;
1901:   ;
1902:L P[587] 1000mm/sec FINE
    :  Arc Start[6]    ;
1903:  Weave Sine[6] ;
1904:L P[588] WELD_SPEED CNT100    ;
1905:L P[592] WELD_SPEED CNT100    ;
1906:L P[593] WELD_SPEED FINE
    :  Arc End[6]    ;
1907:  Weave End ;
1908:   ;
1909:   ;
1910:   ;
1911:J P[534] 50% CNT10    ;
1912:   ;
1913:  !********POSITIONER MOVE******** ;
1914:J P[535] 40% CNT10    ;
1915:   ;
1916:J P[536] 20% CNT5    ;
1917:   ;
1918:L P[537] 1000mm/sec CNT25    ;
1919:   ;
1920:   ;
1921:  !FR50L1730 ;
1922:  IF R[15:TECH HOLD]=1732,CALL TECH_HOLD ;
1923:   ;
1924:   ;
1925:   ;
1926:   ;
1927:L P[594] 1000mm/sec FINE
    :  Arc Start[6]    ;
1928:  Weave Sine[6] ;
1929:  Track TAST[6] ;
1930:L P[599] WELD_SPEED CNT100    ;
1931:L P[600] WELD_SPEED CNT100    ;
1932:L P[601] WELD_SPEED FINE
    :  Arc End[6]    ;
1933:  Weave End ;
1934:  Track End ;
1935:   ;
1936:   ;
1937:   ;
1938:L P[542] 1000mm/sec CNT25    ;
1939:   ;
1940:J P[543] 50% CNT10    ;
1941:   ;
1942:  !********POSITIONER MOVE******** ;
1943:J P[544] 80% CNT10    ;
1944:   ;
1945:   ;
1946:  !FR50L1740 ;
1947:  IF R[15:TECH HOLD]=1742,CALL TECH_HOLD ;
1948:   ;
1949:   ;
1950:   ;
1951:   ;
1952:L P[602] 1000mm/sec FINE
    :  Arc Start[6]    ;
1953:  Weave Sine[6] ;
1954:  Track TAST[6] ;
1955:L P[603] WELD_SPEED FINE
    :  Arc End[6]    ;
1956:  Weave End ;
1957:  Track End ;
1958:   ;
1959:   ;
1960:   ;
1961:L P[547] 1000mm/sec CNT25    ;
1962:   ;
1963:L P[548] 1000mm/sec CNT25    ;
1964:   ;
1965:L P[549] 1000mm/sec CNT25    ;
1966:   ;
1967:   ;
1968:  !FR50L1750 ;
1969:  IF R[15:TECH HOLD]=1752,CALL TECH_HOLD ;
1970:   ;
1971:   ;
1972:   ;
1973:   ;
1974:L P[604] 1000mm/sec FINE
    :  Arc Start[6]    ;
1975:  Weave Sine[6] ;
1976:  Track TAST[6] ;
1977:L P[605] WELD_SPEED CNT100    ;
1978:L P[606] WELD_SPEED FINE
    :  Arc End[6]    ;
1979:  Weave End ;
1980:  Track End ;
1981:   ;
1982:   ;
1983:   ;
1984:L P[553] 1000mm/sec CNT25    ;
1985:   ;
1986:L P[554] 1000mm/sec CNT100    ;
1987:   ;
1988:L P[555] 1000mm/sec CNT100    ;
1989:   ;
1990:J P[508] 50% CNT40    ;
1991:   ;
1992:  CALL HOME    ;
1993:  CALL T_CLEAN    ;
1994:   ;
1995:J P[556] 50% CNT30    ;
1996:   ;
1997:   ;
1998:  !FR50L1770 ;
1999:  IF R[15:TECH HOLD]=1772,CALL TECH_HOLD ;
2000:   ;
2001:   ;
2002:   ;
2003:   ;
2004:L P[609] 1000mm/sec FINE
    :  Arc Start[6]    ;
2005:  Weave Sine[6] ;
2006:  Track TAST[6] ;
2007:L P[610] WELD_SPEED FINE
    :  Arc End[6]    ;
2008:  Weave End ;
2009:  Track End ;
2010:   ;
2011:   ;
2012:   ;
2013:L P[559] 1000mm/sec CNT100    ;
2014:   ;
2015:J P[560] 50% CNT25    ;
2016:   ;
2017:L P[611] 1000mm/sec FINE
    :  Arc Start[6]    ;
2018:  Weave Sine[6] ;
2019:L P[612] WELD_SPEED FINE
    :  Arc End[6]    ;
2020:  Weave End ;
2021:   ;
2022:   ;
2023:L P[563] 1200mm/sec CNT100    ;
2024:   ;
2025:L P[89] 800mm/sec CNT100    ;
2026:   ;
2027:L P[565] 1000mm/sec CNT20    ;
2028:   ;
2029:L P[613] 960mm/sec FINE
    :  Arc Start[6]    ;
2030:  Weave Sine[6] ;
2031:L P[614] WELD_SPEED FINE
    :  Arc End[6]    ;
2032:  Weave End ;
2033:   ;
2034:L P[568] 1000mm/sec CNT25    ;
2035:   ;
2036:J P[569] 50% CNT40    ;
2037:   ;
2038:  !********POSITIONER MOVE******** ;
2039:J P[371] 90% CNT40    ;
2040:   ;
2041:L P[572] 1000mm/sec CNT25    ;
2042:   ;
2043:L P[573] 1000mm/sec CNT25    ;
2044:   ;
2045:   ;
2046:  !FR50L1780 ;
2047:  IF R[15:TECH HOLD]=1782,CALL TECH_HOLD ;
2048:   ;
2049:   ;
2050:   ;
2051:   ;
2052:L P[615] 500mm/sec FINE
    :  Arc Start[6]    ;
2053:  Weave Sine[6] ;
2054:  Track TAST[6] ;
2055:L P[616] WELD_SPEED FINE
    :  Arc End[6]    ;
2056:  Weave End ;
2057:  Track End ;
2058:   ;
2059:   ;
2060:   ;
2061:L P[576] 500mm/sec CNT25    ;
2062:   ;
2063:L P[577] 1000mm/sec CNT25    ;
2064:   ;
2065:  !********POSITIONER MOVE******** ;
2066:J P[578] 90% CNT25    ;
2067:   ;
2068:   ;
2069:  !FR50L1790 ;
2070:  IF R[15:TECH HOLD]=1792,CALL TECH_HOLD ;
2071:   ;
2072:   ;
2073:   ;
2074:   ;
2075:L P[617] 1000mm/sec FINE
    :  Arc Start[6]    ;
2076:  Weave Sine[6] ;
2077:  Track TAST[6] ;
2078:L P[622] WELD_SPEED FINE
    :  Arc End[6]    ;
2079:  Weave End ;
2080:  Track End ;
2081:   ;
2082:   ;
2083:   ;
2084:L P[581] 1000mm/sec CNT100    ;
2085:   ;
2086:   ;
2087:  !FR50L1800 ;
2088:  IF R[15:TECH HOLD]=1802,CALL TECH_HOLD ;
2089:   ;
2090:   ;
2091:   ;
2092:   ;
2093:L P[623] 1000mm/sec FINE
    :  Arc Start[6]    ;
2094:  Weave Sine[6] ;
2095:  Track TAST[6] ;
2096:L P[624] WELD_SPEED CNT100    ;
2097:L P[625] WELD_SPEED FINE
    :  Arc End[6]    ;
2098:  Weave End ;
2099:  Track End ;
2100:   ;
2101:   ;
2102:   ;
2103:L P[585] 1000mm/sec CNT40    ;
2104:   ;
2105:   ;
2106:  !FR50L1810 ;
2107:  IF R[15:TECH HOLD]=1812,CALL TECH_HOLD ;
2108:   ;
2109:   ;
2110:   ;
2111:   ;
2112:L P[628] 1000mm/sec FINE
    :  Arc Start[6]    ;
2113:  Weave Sine[6] ;
2114:  Track TAST[6] ;
2115:L P[629] WELD_SPEED CNT100    ;
2116:L P[631] WELD_SPEED FINE
    :  Arc End[6]    ;
2117:  Weave End ;
2118:  Track End ;
2119:   ;
2120:   ;
2121:   ;
2122:L P[589] 1000mm/sec CNT35    ;
2123:   ;
2124:J P[590] 50% CNT25    ;
2125:   ;
2126:L P[591] 1000mm/sec CNT40    ;
2127:   ;
2128:   ;
2129:  !FR50L1820 ;
2130:  IF R[15:TECH HOLD]=1822,CALL TECH_HOLD ;
2131:   ;
2132:   ;
2133:   ;
2134:   ;
2135:L P[632] 1000mm/sec FINE
    :  Arc Start[6]    ;
2136:  Weave Sine[6] ;
2137:L P[633] WELD_SPEED CNT100    ;
2138:L P[635] WELD_SPEED FINE
    :  Arc End[6]    ;
2139:  Weave End ;
2140:   ;
2141:   ;
2142:   ;
2143:L P[595] 1000mm/sec CNT50    ;
2144:   ;
2145:J P[596] 50% CNT60    ;
2146:   ;
2147:J P[597] 50% CNT40    ;
2148:   ;
2149:L P[598] 1000mm/sec CNT25    ;
2150:   ;
2151:   ;
2152:   ;
2153:  !FR50L1830 ;
2154:  IF R[15:TECH HOLD]=1832,CALL TECH_HOLD ;
2155:   ;
2156:   ;
2157:   ;
2158:   ;
2159:L P[636] 1000mm/sec FINE
    :  Arc Start[6]    ;
2160:  Weave Sine[6] ;
2161:  Track TAST[6] ;
2162:L P[637] WELD_SPEED CNT100    ;
2163:C P[642]
    :  P[643] WELD_SPEED CNT100    ;
2164:L P[644] WELD_SPEED CNT100    ;
2165:C P[649]
    :  P[650] WELD_SPEED CNT100    ;
2166:L P[651] WELD_SPEED FINE
    :  Arc End[6]    ;
2167:  Weave End ;
2168:  Track End ;
2169:   ;
2170:   ;
2171:   ;
2172:L P[607] 1000mm/sec CNT60    ;
2173:   ;
2174:J P[608] 50% CNT50    ;
2175:   ;
2176:   ;
2177:  !FR50L1840 ;
2178:  IF R[15:TECH HOLD]=1842,CALL TECH_HOLD ;
2179:   ;
2180:   ;
2181:   ;
2182:   ;
2183:L P[652] 1000mm/sec FINE
    :  Arc Start[6]    ;
2184:  Weave Sine[6] ;
2185:  Track TAST[6] ;
2186:L P[653] WELD_SPEED CNT100    ;
2187:C P[654]
    :  P[655] WELD_SPEED CNT100    ;
2188:L P[656] WELD_SPEED CNT100    ;
2189:L P[657] WELD_SPEED CNT100    ;
2190:L P[658] WELD_SPEED CNT100    ;
2191:L P[659] WELD_SPEED CNT100    ;
2192:L P[660] WELD_SPEED FINE
    :  Arc End[6]    ;
2193:  Weave End ;
2194:  Track End ;
2195:   ;
2196:   ;
2197:   ;
2198:L P[618] 1000mm/sec CNT25    ;
2199:   ;
2200:J P[619] 50% CNT75    ;
2201:   ;
2202:J P[620] 50% CNT75    ;
2203:   ;
2204:J P[372] 50% CNT80    ;
2205:   ;
2206:L P[621] 1000mm/sec CNT40    ;
2207:   ;
2208:   ;
2209:  !FR50L1850 ;
2210:  IF R[15:TECH HOLD]=1852,CALL TECH_HOLD ;
2211:   ;
2212:   ;
2213:   ;
2214:L P[661] 1000mm/sec FINE
    :  Arc Start[6]    ;
2215:  Weave Sine[6] ;
2216:L P[662] WELD_SPEED CNT100    ;
2217:L P[663] WELD_SPEED CNT100    ;
2218:L P[664] WELD_SPEED FINE
    :  Arc End[6]    ;
2219:  Weave End ;
2220:   ;
2221:   ;
2222:   ;
2223:L P[626] 1000mm/sec CNT90    ;
2224:   ;
2225:L P[627] 1000mm/sec CNT100    ;
2226:   ;
2227:   ;
2228:  !FR50L1860 ;
2229:  IF R[15:TECH HOLD]=1862,CALL TECH_HOLD ;
2230:   ;
2231:   ;
2232:   ;
2233:   ;
2234:L P[665] 1000mm/sec FINE
    :  Arc Start[6]    ;
2235:  Weave Sine[6] ;
2236:  Track TAST[6] ;
2237:L P[666] WELD_SPEED FINE
    :  Arc End[6]    ;
2238:  Weave End ;
2239:  Track End ;
2240:   ;
2241:   ;
2242:   ;
2243:L P[630] 1000mm/sec CNT50    ;
2244:   ;
2245:   ;
2246:  !FR50L1870 ;
2247:  IF R[15:TECH HOLD]=1872,CALL TECH_HOLD ;
2248:   ;
2249:   ;
2250:   ;
2251:   ;
2252:L P[667] 1000mm/sec FINE
    :  Arc Start[6]    ;
2253:  Weave Sine[6] ;
2254:  Track TAST[6] ;
2255:L P[668] WELD_SPEED CNT100    ;
2256:L P[669] WELD_SPEED FINE
    :  Arc End[6]    ;
2257:  Weave End ;
2258:  Track End ;
2259:   ;
2260:   ;
2261:   ;
2262:L P[634] 1000mm/sec CNT60    ;
2263:   ;
2264:   ;
2265:  !FR50L1880 ;
2266:  IF R[15:TECH HOLD]=1882,CALL TECH_HOLD ;
2267:   ;
2268:   ;
2269:   ;
2270:   ;
2271:L P[672] 1000mm/sec FINE
    :  Arc Start[6]    ;
2272:  Weave Sine[6] ;
2273:  Track TAST[6] ;
2274:L P[673] WELD_SPEED CNT100    ;
2275:L P[674] WELD_SPEED FINE
    :  Arc End[6]    ;
2276:  Weave End ;
2277:  Track End ;
2278:   ;
2279:   ;
2280:   ;
2281:L P[373] 1000mm/sec CNT25    ;
2282:   ;
2283:J P[638] 50% CNT25    ;
2284:   ;
2285:J P[641] 50% CNT25    ;
2286:   ;
2287:   ;
2288:  !FR50L1900 ;
2289:  IF R[15:TECH HOLD]=1902,CALL TECH_HOLD ;
2290:   ;
2291:   ;
2292:   ;
2293:   ;
2294:L P[675] 1000mm/sec FINE
    :  Arc Start[6]    ;
2295:  Weave Sine[6] ;
2296:  Track TAST[6] ;
2297:L P[676] WELD_SPEED CNT100    ;
2298:L P[677] WELD_SPEED FINE
    :  Arc End[6]    ;
2299:  Weave End ;
2300:  Track End ;
2301:   ;
2302:   ;
2303:   ;
2304:L P[645] 1000mm/sec CNT40    ;
2305:   ;
2306:J P[87] 50% CNT35    ;
2307:  --eg:Insert g2j2 @-90 Loadstop!!! ;
2308:   ;
2309:  !********POSITIONER MOVE******** ;
2310:J P[106] 85% CNT40    ;
2311:   ;
2312:J P[107] 50% CNT80    ;
2313:   ;
2314:   ;
2315:  !FR50L2010 ;
2316:  IF R[15:TECH HOLD]=2012,CALL TECH_HOLD ;
2317:   ;
2318:L P[108] 1000mm/sec CNT25    ;
2319:   ;
2320:   ;
2321:   ;
2322:L P[761] 1000mm/sec FINE
    :  Arc Start[8]    ;
2323:  Weave Sine[8] ;
2324:L P[762] WELD_SPEED CNT100    ;
2325:C P[763]
    :  P[764] WELD_SPEED CNT100    ;
2326:L P[765] WELD_SPEED CNT100    ;
2327:L P[766] WELD_SPEED CNT100    ;
2328:L P[767] WELD_SPEED CNT100    ;
2329:L P[769] WELD_SPEED FINE
    :  Arc End[8]    ;
2330:  Weave End ;
2331:   ;
2332:   ;
2333:   ;
2334:  CALL ARC_LH_DISABLE_LS(1) ;
2335:   ;
2336:L P[469] 1000mm/sec CNT50    ;
2337:   ;
2338:J P[470] 50% CNT100    ;
2339:   ;
2340:J P[471] 50% CNT70    ;
2341:   ;
2342:J P[472] 50% CNT40    ;
2343:   ;
2344:  --eg:Insert g2j2 @-90 Loadstop!!! ;
2345:   ;
2346:  !********POSITIONER MOVE******** ;
2347:J P[118] 85% CNT40    ;
2348:   ;
2349:J P[646] 90% CNT50    ;
2350:   ;
2351:L P[647] 1000mm/sec CNT40    ;
2352:   ;
2353:L P[648] 1000mm/sec CNT25    ;
2354:   ;
2355:   ;
2356:  !FR50L1910 ;
2357:  IF R[15:TECH HOLD]=1912,CALL TECH_HOLD ;
2358:   ;
2359:   ;
2360:   ;
2361:   ;
2362:L P[678] 1000mm/sec FINE
    :  Arc Start[6]    ;
2363:  Weave Sine[6] ;
2364:  Track TAST[6] ;
2365:L P[686] WELD_SPEED CNT100    ;
2366:C P[687]
    :  P[691] WELD_SPEED CNT100    ;
2367:L P[692] WELD_SPEED CNT100    ;
2368:L P[693] WELD_SPEED CNT100    ;
2369:L P[696] WELD_SPEED CNT100    ;
2370:L P[697] WELD_SPEED CNT100    ;
2371:C P[703]
    :  P[704] WELD_SPEED CNT100    ;
2372:L P[705] WELD_SPEED CNT100    ;
2373:C P[706]
    :  P[707] WELD_SPEED CNT100    ;
2374:L P[709] WELD_SPEED CNT100    ;
2375:C P[715]
    :  P[716] WELD_SPEED CNT100    ;
2376:L P[717] WELD_SPEED CNT100    ;
2377:L P[718] WELD_SPEED CNT100    ;
2378:L P[719] WELD_SPEED CNT100    ;
2379:C P[722]
    :  P[723] WELD_SPEED FINE
    :  Arc End[6]    ;
2380:  Weave End ;
2381:  Track End ;
2382:   ;
2383:   ;
2384:L P[670] 1000mm/sec CNT25    ;
2385:   ;
2386:L P[671] 500mm/sec CNT25    ;
2387:   ;
2388:   ;
2389:  !FR50L1911 ;
2390:  IF R[15:TECH HOLD]=1913,CALL TECH_HOLD ;
2391:   ;
2392:   ;
2393:L P[786] 500mm/sec FINE
    :  Arc Start[6]    ;
2394:  Weave Sine[6] ;
2395:  Track TAST[6] ;
2396:L P[787] WELD_SPEED CNT100    ;
2397:C P[788]
    :  P[789] WELD_SPEED CNT100    ;
2398:L P[790] WELD_SPEED CNT100    ;
2399:C P[791]
    :  P[792] WELD_SPEED FINE
    :  Arc End[6]    ;
2400:  Weave End ;
2401:  Track End ;
2402:   ;
2403:L P[679] 1000mm/sec CNT80    ;
2404:   ;
2405:L P[680] 900mm/sec CNT30 Wjnt    ;
2406:   ;
2407:J P[95] 50% CNT90    ;
2408:   ;
2409:J P[681] 50% CNT40    ;
2410:   ;
2411:  !HOME ;
2412:J P[94] 80% CNT40    ;
2413:   ;
2414:  !********POSITIONER MOVE******** ;
2415:J P[682] 90% CNT30    ;
2416:   ;
2417:J P[683] 50% CNT85    ;
2418:   ;
2419:J P[684] 50% CNT30    ;
2420:   ;
2421:L P[685] 1000mm/sec CNT25    ;
2422:   ;
2423:  !TO SKIP FRONT BUMPER WELDS ;
2424:  CALL ARC_DISABLE_FRONT_BMPR_LRG(0) ;
2425:   ;
2426:  !FR50L1920 ;
2427:  IF R[15:TECH HOLD]=1922,CALL TECH_HOLD ;
2428:   ;
2429:  UALM[20] ;
2430:  --eg:CHECK NEXT 3 WELDS ;
2431:   ;
2432:   ;
2433:   ;
2434:L P[731] 1000mm/sec FINE
    :  Arc Start[6]    ;
2435:  Weave Sine[6] ;
2436:  Track TAST[6] ;
2437:L P[734] WELD_SPEED FINE
    :  Arc End[6]    ;
2438:  Weave End ;
2439:  Track End ;
2440:   ;
2441:   ;
2442:   ;
2443:L P[688] 1000mm/sec CNT100    ;
2444:   ;
2445:J P[689] 50% CNT25    ;
2446:   ;
2447:L P[690] 1000mm/sec CNT25    ;
2448:   ;
2449:   ;
2450:  !FR50L1930 ;
2451:  IF R[15:TECH HOLD]=1932,CALL TECH_HOLD ;
2452:   ;
2453:   ;
2454:L P[735] 1000mm/sec FINE
    :  Arc Start[6]    ;
2455:  Weave Sine[6] ;
2456:  Track TAST[6] ;
2457:L P[736] WELD_SPEED CNT100    ;
2458:L P[737] WELD_SPEED FINE
    :  Arc End[6]    ;
2459:  Weave End ;
2460:  Track End ;
2461:   ;
2462:   ;
2463:   ;
2464:L P[694] 1000mm/sec CNT90    ;
2465:   ;
2466:J P[695] 50% CNT40    ;
2467:   ;
2468:   ;
2469:  !FR50L1940 ;
2470:  IF R[15:TECH HOLD]=1942,CALL TECH_HOLD ;
2471:   ;
2472:   ;
2473:   ;
2474:   ;
2475:L P[741] 1000mm/sec FINE
    :  Arc Start[6]    ;
2476:  Weave Sine[6] ;
2477:  Track TAST[6] ;
2478:L P[742] WELD_SPEED FINE
    :  Arc End[6]    ;
2479:  Weave End ;
2480:  Track End ;
2481:   ;
2482:   ;
2483:   ;
2484:  CALL ARC_DISABLE_FRONT_BMPR_LRG(1) ;
2485:   ;
2486:L P[698] 1000mm/sec CNT25    ;
2487:   ;
2488:J P[699] 50% CNT40    ;
2489:   ;
2490:  !********POSITIONER MOVE******** ;
2491:J P[700] 90% CNT30    ;
2492:   ;
2493:J P[701] 50% CNT30    ;
2494:   ;
2495:   ;
2496:  CALL ARC_LH_DISABLE_LS(0) ;
2497:   ;
2498:  !FR50L1950 ;
2499:  IF R[15:TECH HOLD]=1952,CALL TECH_HOLD ;
2500:   ;
2501:   ;
2502:L P[702] 1000mm/sec CNT25    ;
2503:   ;
2504:   ;
2505:   ;
2506:L P[743] 1000mm/sec FINE
    :  Arc Start[6]    ;
2507:  Weave Sine[6] ;
2508:  Track TAST[6] ;
2509:L P[744] WELD_SPEED CNT100    ;
2510:L P[745] WELD_SPEED CNT100    ;
2511:C P[746]
    :  P[747] WELD_SPEED FINE
    :  Arc End[6]    ;
2512:  Weave End ;
2513:  Track End ;
2514:   ;
2515:   ;
2516:   ;
2517:  CALL ARC_LH_DISABLE_LS(1) ;
2518:   ;
2519:L P[708] 1000mm/sec CNT50    ;
2520:   ;
2521:J P[97] 50% CNT25    ;
2522:   ;
2523:J P[710] 50% CNT25    ;
2524:   ;
2525:  !********POSITIONER MOVE******** ;
2526:J P[2] 85% CNT40    ;
2527:   ;
2528:J P[105] 50% CNT25    ;
2529:   ;
2530:L P[113] 1000mm/sec CNT25    ;
2531:   ;
2532:  CALL ARC_DISABLE_RH_LS(0) ;
2533:   ;
2534:  !FR50L1970 ;
2535:  IF R[15:TECH HOLD]=1972,CALL TECH_HOLD ;
2536:   ;
2537:   ;
2538:   ;
2539:   ;
2540:L P[753] 800mm/sec FINE
    :  Arc Start[6]    ;
2541:  Weave Sine[6] ;
2542:  Track TAST[6] ;
2543:L P[754] WELD_SPEED CNT100    ;
2544:C P[755]
    :  P[756] WELD_SPEED FINE
    :  Arc End[6]    ;
2545:  Track End ;
2546:  Weave End ;
2547:   ;
2548:   ;
2549:   ;
2550:L P[564] 800mm/sec CNT5    ;
2551:   ;
2552:J P[571] 20% CNT40    ;
2553:   ;
2554:J P[639] 40% CNT25    ;
2555:   ;
2556:J P[640] 75% CNT50    ;
2557:   ;
2558:  !********POSITIONER MOVE******** ;
2559:J P[711] 85% CNT30    ;
2560:   ;
2561:J P[712] 50% CNT80    ;
2562:   ;
2563:L P[713] 1000mm/sec CNT40    ;
2564:   ;
2565:   ;
2566:  !FR50L1960 ;
2567:  IF R[15:TECH HOLD]=1962,CALL TECH_HOLD ;
2568:   ;
2569:   ;
2570:L P[714] 500mm/sec CNT25    ;
2571:   ;
2572:   ;
2573:   ;
2574:L P[748] 1000mm/sec FINE
    :  Arc Start[6]    ;
2575:  Weave Sine[6] ;
2576:  Track TAST[6] ;
2577:L P[749] WELD_SPEED CNT100    ;
2578:L P[750] WELD_SPEED CNT100    ;
2579:C P[751]
    :  P[752] WELD_SPEED FINE
    :  Arc End[6]    ;
2580:  Weave End ;
2581:  Track End ;
2582:   ;
2583:   ;
2584:   ;
2585:  CALL ARC_DISABLE_RH_LS(1) ;
2586:   ;
2587:L P[720] 500mm/sec CNT35    ;
2588:   ;
2589:L P[721] 1000mm/sec CNT100    ;
2590:   ;
2591:J P[99] 100% CNT30    ;
2592:   ;
2593:  !******** POSITIONER MOVE ******* ;
2594:J P[793] 85% CNT30    ;
2595:   ;
2596:J P[732] 75% CNT25    ;
2597:   ;
2598:L P[733] 1000mm/sec CNT100    ;
2599:   ;
2600:   ;
2601:  CALL ARC_LH_DISABLE_LS(0) ;
2602:   ;
2603:  !FR50L1980 ;
2604:  IF R[15:TECH HOLD]=1982,CALL TECH_HOLD ;
2605:   ;
2606:   ;
2607:   ;
2608:   ;
2609:L P[757] 800mm/sec FINE
    :  Arc Start[6]    ;
2610:  Weave Sine[6] ;
2611:  Track TAST[6] ;
2612:L P[758] WELD_SPEED CNT100    ;
2613:C P[759]
    :  P[760] WELD_SPEED FINE
    :  Arc End[6]    ;
2614:  Weave End ;
2615:  Track End ;
2616:   ;
2617:   ;
2618:   ;
2619:L P[738] 800mm/sec CNT20    ;
2620:   ;
2621:L P[739] 1000mm/sec CNT100    ;
2622:   ;
2623:J P[740] 100% CNT100    ;
2624:   ;
2625:  !HOME ;
2626:J P[104] 100% CNT30    ;
2627:   ;
2628:  CALL HOME    ;
2629:   ;
2630:  !********POSITIONER MOVE******** ;
2631:  CALL LOAD_POS    ;
2632:   ;
2633:  R[79:TEST LRG WELDDIT]=($AWEPRODSTAT[1].$WELD_DIST) ;
2634:  !11111111111111111111111111111111 ;
/POS
P[1]{
   GP1:
	UF : 1, UT : 1,		CONFIG : 'N U T, 0, 0, 0',
	X =  1048.285  mm,	Y = -1294.070  mm,	Z =   701.250  mm,
	W =     -.009 deg,	P =    41.863 deg,	R =  -150.867 deg
   GP2:
	UF : 1, UT : 1,
	J1=     0.000 deg,	J2=   -40.000 deg
};
P[2]{
   GP1:
	UF : 1, UT : 1,		CONFIG : 'N U T, 0, 0, 0',
	X =  1171.584  mm,	Y = -1326.619  mm,	Z =  1560.411  mm,
	W =   -31.995 deg,	P =   -11.977 deg,	R =    17.020 deg
   GP2:
	UF : 1, UT : 1,
	J1=   180.000 deg,	J2=  -125.000 deg
};
P[3]{
   GP1:
	UF : 1, UT : 1,		CONFIG : 'N U T, 0, 0, 0',
	X =  1209.555  mm,	Y = -1322.972  mm,	Z =   229.179  mm,
	W =     -.010 deg,	P =    41.970 deg,	R =  -145.526 deg
   GP2:
	UF : 1, UT : 1,
	J1=     0.000 deg,	J2=   -40.000 deg
};
P[4]{
   GP1:
	UF : 1, UT : 1,		CONFIG : 'N U B, 0, 0, 0',
	X =   356.032  mm,	Y =    -2.146  mm,	Z =  2424.050  mm,
	W =      .001 deg,	P =   -40.002 deg,	R =     -.005 deg
   GP2:
	UF : 1, UT : 1,
	J1=     0.000 deg,	J2=   -40.000 deg
};
P[5]{
   GP1:
	UF : 1, UT : 1,		CONFIG : 'N U T, 0, 0, 0',
	X =  1252.058  mm,	Y = -1261.378  mm,	Z =    72.461  mm,
	W =    -1.699 deg,	P =    44.143 deg,	R =  -145.630 deg
   GP2:
	UF : 1, UT : 1,
	J1=     0.000 deg,	J2=   -40.000 deg
};
P[6]{
   GP1:
	UF : 1, UT : 1,		CONFIG : 'N U T, 0, 0, 0',
	X =  1307.345  mm,	Y = -1320.375  mm,	Z =    70.982  mm,
	W =     1.500 deg,	P =    44.727 deg,	R =  -177.468 deg
   GP2:
	UF : 1, UT : 1,
	J1=     0.000 deg,	J2=   -40.000 deg
};
P[7]{
   GP1:
	UF : 1, UT : 1,		CONFIG : 'N U B, 0, 0, 0',
	X =   356.032  mm,	Y =    -2.146  mm,	Z =  2424.049  mm,
	W =      .001 deg,	P =   -40.002 deg,	R =     -.005 deg
   GP2:
	UF : 1, UT : 1,
	J1=    45.000 deg,	J2=     0.000 deg
};
P[8]{
   GP1:
	UF : 1, UT : 1,		CONFIG : 'N U T, 0, 0, 0',
	X =  1272.049  mm,	Y = -1319.952  mm,	Z =   170.275  mm,
	W =    -4.003 deg,	P =    44.859 deg,	R =  -166.486 deg
   GP2:
	UF : 1, UT : 1,
	J1=     0.000 deg,	J2=   -40.000 deg
};
P[9]{
   GP1:
	UF : 1, UT : 1,		CONFIG : 'N U T, 0, 0, 0',
	X =   909.960  mm,	Y =  -872.839  mm,	Z =   170.274  mm,
	W =      .297 deg,	P =    44.999 deg,	R =  -138.174 deg
   GP2:
	UF : 1, UT : 1,
	J1=     0.000 deg,	J2=   -40.000 deg
};
P[10]{
   GP1:
	UF : 1, UT : 1,		CONFIG : 'N U T, 0, 0, 0',
	X =   902.346  mm,	Y =  -835.521  mm,	Z =    69.924  mm,
	W =      .907 deg,	P =    42.840 deg,	R =  -137.766 deg
   GP2:
	UF : 1, UT : 1,
	J1=     0.000 deg,	J2=   -40.000 deg
};
P[11]{
   GP1:
	UF : 1, UT : 1,		CONFIG : 'N U T, 0, 0, 0',
	X =  1236.294  mm,	Y = -1234.316  mm,	Z =    69.654  mm,
	W =      .456 deg,	P =    44.458 deg,	R =  -141.251 deg
   GP2:
	UF : 1, UT : 1,
	J1=     0.000 deg,	J2=   -40.000 deg
};
P[12]{
   GP1:
	UF : 1, UT : 1,		CONFIG : 'N U T, 0, 0, 0',
	X =  1163.391  mm,	Y = -1298.112  mm,	Z =   230.228  mm,
	W =     1.291 deg,	P =    44.986 deg,	R =  -138.174 deg
   GP2:
	UF : 1, UT : 1,
	J1=     0.000 deg,	J2=   -40.000 deg
};
P[13]{
   GP1:
	UF : 1, UT : 1,		CONFIG : 'N U T, 0, 0, 0',
	X =   860.828  mm,	Y =  -857.112  mm,	Z =   230.228  mm,
	W =     1.291 deg,	P =    44.986 deg,	R =  -138.174 deg
   GP2:
	UF : 1, UT : 1,
	J1=     0.000 deg,	J2=   -40.000 deg
};
P[14]{
   GP1:
	UF : 1, UT : 1,		CONFIG : 'N U T, 0, 0, 0',
	X =   872.611  mm,	Y =  -807.728  mm,	Z =    71.519  mm,
	W =    -2.028 deg,	P =    42.190 deg,	R =  -140.469 deg
   GP2:
	UF : 1, UT : 1,
	J1=     0.000 deg,	J2=   -40.000 deg
};
P[15]{
   GP1:
	UF : 1, UT : 1,		CONFIG : 'N U T, 0, 0, 0',
	X =   825.707  mm,	Y =  -749.978  mm,	Z =    70.668  mm,
	W =    -1.995 deg,	P =    42.640 deg,	R =  -109.079 deg
   GP2:
	UF : 1, UT : 1,
	J1=     0.000 deg,	J2=   -40.000 deg
};
P[16]{
   GP1:
	UF : 1, UT : 1,		CONFIG : 'N U T, 0, 0, 0',
	X =   643.854  mm,	Y = -1045.560  mm,	Z =   456.782  mm,
	W =     1.290 deg,	P =    44.986 deg,	R =  -124.491 deg
   GP2:
	UF : 1, UT : 1,
	J1=     0.000 deg,	J2=   -40.000 deg
};
P[17]{
   GP1:
	UF : 1, UT : 1,		CONFIG : 'N U T, 0, 0, 0',
	X =   908.243  mm,	Y =     -.972  mm,	Z =  2177.323  mm,
	W =     -.010 deg,	P =   -45.000 deg,	R =     0.000 deg
   GP2:
	UF : 1, UT : 1,
	J1=    90.000 deg,	J2=     0.000 deg
};
P[18]{
   GP1:
	UF : 1, UT : 1,		CONFIG : 'N U T, 0, 0, 0',
	X =  1593.884  mm,	Y =    54.651  mm,	Z =  1425.564  mm,
	W =    40.560 deg,	P =     2.984 deg,	R =   -28.829 deg
   GP2:
	UF : 1, UT : 1,
	J1=    90.000 deg,	J2=     0.000 deg
};
P[19]{
   GP1:
	UF : 1, UT : 1,		CONFIG : 'N U T, 0, 0, 0',
	X =  2419.244  mm,	Y =   170.457  mm,	Z =   756.322  mm,
	W =    40.554 deg,	P =     2.977 deg,	R =   -28.823 deg
   GP2:
	UF : 1, UT : 1,
	J1=    90.000 deg,	J2=     0.000 deg
};
P[20]{
   GP1:
	UF : 1, UT : 1,		CONFIG : 'N U T, 0, 0, 0',
	X =  2486.244  mm,	Y =   320.457  mm,	Z =   579.520  mm,
	W =    40.554 deg,	P =     2.977 deg,	R =    -7.352 deg
   GP2:
	UF : 1, UT : 1,
	J1=    90.000 deg,	J2=     0.000 deg
};
P[21]{
   GP1:
	UF : 1, UT : 1,		CONFIG : 'N U T, 0, 0, 0',
	X =  2508.188  mm,	Y =   408.450  mm,	Z =   487.642  mm,
	W =    44.781 deg,	P =     5.019 deg,	R =    -1.188 deg
   GP2:
	UF : 1, UT : 1,
	J1=    90.000 deg,	J2=     0.000 deg
};
P[22]{
   GP1:
	UF : 1, UT : 1,		CONFIG : 'N U T, 0, 0, 0',
	X =  2466.409  mm,	Y =   408.572  mm,	Z =   487.702  mm,
	W =    44.791 deg,	P =     5.023 deg,	R =    -1.193 deg
   GP2:
	UF : 1, UT : 1,
	J1=    90.000 deg,	J2=     0.000 deg
};
P[23]{
   GP1:
	UF : 1, UT : 1,		CONFIG : 'N U T, 0, 0, 0',
	X =  2443.024  mm,	Y =   407.813  mm,	Z =   489.461  mm,
	W =    44.788 deg,	P =     5.020 deg,	R =    30.075 deg
   GP2:
	UF : 1, UT : 1,
	J1=    90.000 deg,	J2=     0.000 deg
};
P[24]{
   GP1:
	UF : 1, UT : 1,		CONFIG : 'N U T, 0, 0, 0',
	X =  2521.819  mm,	Y =   261.320  mm,	Z =   656.993  mm,
	W =    44.759 deg,	P =     5.240 deg,	R =    21.047 deg
   GP2:
	UF : 1, UT : 1,
	J1=    90.000 deg,	J2=     0.000 deg
};
P[25]{
   GP1:
	UF : 1, UT : 1,		CONFIG : 'N U T, 0, 0, 0',
	X =  2511.367  mm,	Y =  -251.873  mm,	Z =   577.119  mm,
	W =   -39.345 deg,	P =     9.413 deg,	R =    11.283 deg
   GP2:
	UF : 1, UT : 1,
	J1=    90.000 deg,	J2=     0.000 deg
};
P[26]{
   GP1:
	UF : 1, UT : 1,		CONFIG : 'N U T, 0, 0, 0',
	X =  2524.947  mm,	Y =  -411.523  mm,	Z =   487.782  mm,
	W =   -44.055 deg,	P =    10.311 deg,	R =     9.166 deg
   GP2:
	UF : 1, UT : 1,
	J1=    90.000 deg,	J2=     0.000 deg
};
P[27]{
   GP1:
	UF : 1, UT : 1,		CONFIG : 'N U T, 0, 0, 0',
	X =  2481.308  mm,	Y =  -411.463  mm,	Z =   487.996  mm,
	W =   -44.053 deg,	P =    10.307 deg,	R =     9.166 deg
   GP2:
	UF : 1, UT : 1,
	J1=    90.000 deg,	J2=     0.000 deg
};
P[28]{
   GP1:
	UF : 1, UT : 1,		CONFIG : 'N U T, 0, 0, 0',
	X =  2449.567  mm,	Y =  -411.710  mm,	Z =   486.469  mm,
	W =   -44.056 deg,	P =    10.309 deg,	R =   -21.686 deg
   GP2:
	UF : 1, UT : 1,
	J1=    90.000 deg,	J2=     0.000 deg
};
P[29]{
   GP1:
	UF : 1, UT : 1,		CONFIG : 'N U T, 0, 0, 0',
	X =  2549.787  mm,	Y =  -262.671  mm,	Z =   682.477  mm,
	W =   -44.052 deg,	P =    10.305 deg,	R =   -20.066 deg
   GP2:
	UF : 1, UT : 1,
	J1=    90.000 deg,	J2=     0.000 deg
};
P[30]{
   GP1:
	UF : 1, UT : 1,		CONFIG : 'N U T, 0, 0, 0',
	X =  2103.073  mm,	Y =   282.472  mm,	Z =   462.977  mm,
	W =    30.589 deg,	P =    34.770 deg,	R =    43.796 deg
   GP2:
	UF : 1, UT : 1,
	J1=    90.000 deg,	J2=     0.000 deg
};
P[31]{
   GP1:
	UF : 1, UT : 1,		CONFIG : 'N U T, 0, 0, 0',
	X =  2009.910  mm,	Y =   392.326  mm,	Z =   357.903  mm,
	W =    43.297 deg,	P =    13.770 deg,	R =    75.808 deg
   GP2:
	UF : 1, UT : 1,
	J1=    90.000 deg,	J2=     0.000 deg
};
P[32]{
   GP1:
	UF : 1, UT : 1,		CONFIG : 'N U T, 0, 0, 0',
	X =  2009.910  mm,	Y =   312.166  mm,	Z =   357.903  mm,
	W =    43.297 deg,	P =    13.770 deg,	R =    75.808 deg
   GP2:
	UF : 1, UT : 1,
	J1=    90.000 deg,	J2=     0.000 deg
};
P[33]{
   GP1:
	UF : 1, UT : 1,		CONFIG : 'N U T, 0, 0, 0',
	X =  2084.488  mm,	Y =   314.464  mm,	Z =   441.765  mm,
	W =    43.281 deg,	P =    13.759 deg,	R =    75.826 deg
   GP2:
	UF : 1, UT : 1,
	J1=    90.000 deg,	J2=     0.000 deg
};
P[34]{
   GP1:
	UF : 1, UT : 1,		CONFIG : 'N U T, 0, 0, 0',
	X =  2086.988  mm,	Y =  -331.633  mm,	Z =   441.764  mm,
	W =   -41.228 deg,	P =    19.917 deg,	R =   -68.756 deg
   GP2:
	UF : 1, UT : 1,
	J1=    90.000 deg,	J2=     0.000 deg
};
P[35]{
   GP1:
	UF : 1, UT : 1,		CONFIG : 'N U T, 0, 0, 0',
	X =  2009.490  mm,	Y =  -404.811  mm,	Z =   359.074  mm,
	W =   -41.229 deg,	P =    19.917 deg,	R =   -68.757 deg
   GP2:
	UF : 1, UT : 1,
	J1=    90.000 deg,	J2=     0.000 deg
};
P[36]{
   GP1:
	UF : 1, UT : 1,		CONFIG : 'N U T, 0, 0, 0',
	X =  2009.489  mm,	Y =  -322.731  mm,	Z =   359.074  mm,
	W =   -41.229 deg,	P =    19.917 deg,	R =   -68.757 deg
   GP2:
	UF : 1, UT : 1,
	J1=    90.000 deg,	J2=     0.000 deg
};
P[37]{
   GP1:
	UF : 1, UT : 1,		CONFIG : 'N U T, 0, 0, 0',
	X =  2106.807  mm,	Y =  -322.474  mm,	Z =   465.914  mm,
	W =   -41.228 deg,	P =    19.917 deg,	R =   -68.756 deg
   GP2:
	UF : 1, UT : 1,
	J1=    90.000 deg,	J2=     0.000 deg
};
P[38]{
   GP1:
	UF : 1, UT : 1,		CONFIG : 'N U T, 0, 0, 0',
	X =  2109.307  mm,	Y =    75.081  mm,	Z =   465.913  mm,
	W =     3.207 deg,	P =    44.910 deg,	R =   -85.462 deg
   GP2:
	UF : 1, UT : 1,
	J1=    90.000 deg,	J2=     0.000 deg
};
P[39]{
   GP1:
	UF : 1, UT : 1,		CONFIG : 'N U T, 0, 0, 0',
	X =  2681.306  mm,	Y =  -103.919  mm,	Z =  -438.087  mm,
	W =    -1.257 deg,	P =    33.277 deg,	R =   -88.589 deg
   GP2:
	UF : 1, UT : 1,
	J1=    90.000 deg,	J2=     0.000 deg
};
P[40]{
   GP1:
	UF : 1, UT : 1,		CONFIG : 'N U T, 0, 0, 0',
	X =  2736.558  mm,	Y =   -56.451  mm,	Z =  -598.484  mm,
	W =      .970 deg,	P =    44.992 deg,	R =   -88.628 deg
   GP2:
	UF : 1, UT : 1,
	J1=    90.000 deg,	J2=     0.000 deg
};
P[41]{
   GP1:
	UF : 1, UT : 1,		CONFIG : 'N U T, 0, 0, 0',
	X =  2767.036  mm,	Y =   -56.451  mm,	Z =  -598.486  mm,
	W =      .970 deg,	P =    44.992 deg,	R =   -88.628 deg
   GP2:
	UF : 1, UT : 1,
	J1=    90.000 deg,	J2=     0.000 deg
};
P[42]{
   GP1:
	UF : 1, UT : 1,		CONFIG : 'N U T, 0, 0, 0',
	X =  2676.306  mm,	Y =  -106.919  mm,	Z =  -439.087  mm,
	W =    -1.257 deg,	P =    33.277 deg,	R =   -88.589 deg
   GP2:
	UF : 1, UT : 1,
	J1=    90.000 deg,	J2=     0.000 deg
};
P[43]{
   GP1:
	UF : 1, UT : 1,		CONFIG : 'N U T, 0, 0, 0',
	X =  2576.306  mm,	Y =    -6.919  mm,	Z =  -439.087  mm,
	W =    -1.257 deg,	P =    33.277 deg,	R =   -88.589 deg
   GP2:
	UF : 1, UT : 1,
	J1=    90.000 deg,	J2=     0.000 deg
};
P[44]{
   GP1:
	UF : 1, UT : 1,		CONFIG : 'N U T, 0, 0, 0',
	X =  2582.224  mm,	Y =   118.706  mm,	Z =  -400.809  mm,
	W =      .677 deg,	P =    39.803 deg,	R =    91.170 deg
   GP2:
	UF : 1, UT : 1,
	J1=    90.000 deg,	J2=     0.000 deg
};
P[45]{
   GP1:
	UF : 1, UT : 1,		CONFIG : 'N U T, 0, 0, 0',
	X =  2706.224  mm,	Y =   118.706  mm,	Z =  -483.809  mm,
	W =      .677 deg,	P =    39.803 deg,	R =    91.170 deg
   GP2:
	UF : 1, UT : 1,
	J1=    90.000 deg,	J2=     0.000 deg
};
P[46]{
   GP1:
	UF : 1, UT : 1,		CONFIG : 'N U T, 0, 0, 0',
	X =  2737.214  mm,	Y =    52.045  mm,	Z =  -596.220  mm,
	W =      .898 deg,	P =    44.994 deg,	R =    91.270 deg
   GP2:
	UF : 1, UT : 1,
	J1=    90.000 deg,	J2=     0.000 deg
};
P[47]{
   GP1:
	UF : 1, UT : 1,		CONFIG : 'N U T, 0, 0, 0',
	X =  2765.224  mm,	Y =    53.223  mm,	Z =  -596.928  mm,
	W =      .899 deg,	P =    44.991 deg,	R =    91.266 deg
   GP2:
	UF : 1, UT : 1,
	J1=    90.000 deg,	J2=     0.000 deg
};
P[48]{
   GP1:
	UF : 1, UT : 1,		CONFIG : 'N U T, 0, 0, 0',
	X =  2706.224  mm,	Y =   118.706  mm,	Z =  -483.809  mm,
	W =      .677 deg,	P =    39.803 deg,	R =    91.170 deg
   GP2:
	UF : 1, UT : 1,
	J1=    90.000 deg,	J2=     0.000 deg
};
P[49]{
   GP1:
	UF : 1, UT : 1,		CONFIG : 'N U T, 0, 0, 0',
	X =  2750.938  mm,	Y =   112.285  mm,	Z =  -474.250  mm,
	W =     -.713 deg,	P =    25.922 deg,	R =     -.241 deg
   GP2:
	UF : 1, UT : 1,
	J1=    90.000 deg,	J2=     0.000 deg
};
P[50]{
   GP1:
	UF : 1, UT : 1,		CONFIG : 'N U T, 0, 0, 0',
	X =  2778.081  mm,	Y =    53.285  mm,	Z =  -487.998  mm,
	W =     -.713 deg,	P =    25.922 deg,	R =     -.241 deg
   GP2:
	UF : 1, UT : 1,
	J1=    90.000 deg,	J2=     0.000 deg
};
P[51]{
   GP1:
	UF : 1, UT : 1,		CONFIG : 'N U T, 0, 0, 0',
	X =  2771.547  mm,	Y =    44.594  mm,	Z =  -599.203  mm,
	W =     -.289 deg,	P =    37.601 deg,	R =      .738 deg
   GP2:
	UF : 1, UT : 1,
	J1=    90.000 deg,	J2=     0.000 deg
};
P[52]{
   GP1:
	UF : 1, UT : 1,		CONFIG : 'N U T, 0, 0, 0',
	X =  2771.146  mm,	Y =   -56.494  mm,	Z =  -598.357  mm,
	W =     -.293 deg,	P =    37.601 deg,	R =      .748 deg
   GP2:
	UF : 1, UT : 1,
	J1=    90.000 deg,	J2=     0.000 deg
};
P[53]{
   GP1:
	UF : 1, UT : 1,		CONFIG : 'N U T, 0, 0, 0',
	X =  2774.367  mm,	Y =   -45.046  mm,	Z =  -326.584  mm,
	W =     -.063 deg,	P =     6.406 deg,	R =     -.319 deg
   GP2:
	UF : 1, UT : 1,
	J1=    90.000 deg,	J2=     0.000 deg
};
P[54]{
   GP1:
	UF : 1, UT : 1,		CONFIG : 'N U T, 0, 0, 0',
	X =  2318.510  mm,	Y =     4.126  mm,	Z =   836.416  mm,
	W =     -.063 deg,	P =     6.406 deg,	R =     -.319 deg
   GP2:
	UF : 1, UT : 1,
	J1=    90.000 deg,	J2=     0.000 deg
};
P[55]{
   GP1:
	UF : 1, UT : 1,		CONFIG : 'N U T, 0, 0, 0',
	X =  2651.064  mm,	Y =   274.146  mm,	Z =   596.222  mm,
	W =    40.438 deg,	P =    -1.956 deg,	R =     2.337 deg
   GP2:
	UF : 1, UT : 1,
	J1=    90.000 deg,	J2=     0.000 deg
};
P[56]{
   GP1:
	UF : 1, UT : 1,		CONFIG : 'N U T, 0, 0, 0',
	X =  2678.366  mm,	Y =   323.391  mm,	Z =   552.416  mm,
	W =    40.027 deg,	P =    -6.599 deg,	R =     7.835 deg
   GP2:
	UF : 1, UT : 1,
	J1=    90.000 deg,	J2=     0.000 deg
};
P[57]{
   GP1:
	UF : 1, UT : 1,		CONFIG : 'N U T, 0, 0, 0',
	X =  2751.342  mm,	Y =   410.859  mm,	Z =   451.447  mm,
	W =    44.538 deg,	P =    -7.208 deg,	R =     7.272 deg
   GP2:
	UF : 1, UT : 1,
	J1=    90.000 deg,	J2=     0.000 deg
};
P[58]{
   GP1:
	UF : 1, UT : 1,		CONFIG : 'N U T, 0, 0, 0',
	X =  2710.782  mm,	Y =   408.789  mm,	Z =   452.225  mm,
	W =    44.541 deg,	P =    -7.214 deg,	R =     7.272 deg
   GP2:
	UF : 1, UT : 1,
	J1=    90.000 deg,	J2=     0.000 deg
};
P[59]{
   GP1:
	UF : 1, UT : 1,		CONFIG : 'N U T, 0, 0, 0',
	X =  2698.437  mm,	Y =   269.508  mm,	Z =   599.906  mm,
	W =    44.541 deg,	P =    -7.214 deg,	R =     7.272 deg
   GP2:
	UF : 1, UT : 1,
	J1=    90.000 deg,	J2=     0.000 deg
};
P[60]{
   GP1:
	UF : 1, UT : 1,		CONFIG : 'N U T, 0, 0, 0',
	X =  2703.937  mm,	Y =  -282.492  mm,	Z =   602.906  mm,
	W =   -34.404 deg,	P =     5.822 deg,	R =     8.425 deg
   GP2:
	UF : 1, UT : 1,
	J1=    90.000 deg,	J2=     0.000 deg
};
P[61]{
   GP1:
	UF : 1, UT : 1,		CONFIG : 'N U T, 0, 0, 0',
	X =  2754.725  mm,	Y =  -417.352  mm,	Z =   456.544  mm,
	W =   -44.517 deg,	P =     7.212 deg,	R =     7.270 deg
   GP2:
	UF : 1, UT : 1,
	J1=    90.000 deg,	J2=     0.000 deg
};
P[62]{
   GP1:
	UF : 1, UT : 1,		CONFIG : 'N U T, 0, 0, 0',
	X =  2716.537  mm,	Y =  -417.597  mm,	Z =   455.165  mm,
	W =   -44.526 deg,	P =     7.207 deg,	R =     7.276 deg
   GP2:
	UF : 1, UT : 1,
	J1=    90.000 deg,	J2=     0.000 deg
};
P[63]{
   GP1:
	UF : 1, UT : 1,		CONFIG : 'N U T, 0, 0, 0',
	X =  2699.988  mm,	Y =  -282.600  mm,	Z =   597.231  mm,
	W =   -44.541 deg,	P =     7.214 deg,	R =     7.272 deg
   GP2:
	UF : 1, UT : 1,
	J1=    90.000 deg,	J2=     0.000 deg
};
P[64]{
   GP1:
	UF : 1, UT : 1,		CONFIG : 'F U T, 0, 0, 0',
	X =  2542.011  mm,	Y =    62.997  mm,	Z =   733.500  mm,
	W =      .337 deg,	P =   -50.731 deg,	R =     6.061 deg
   GP2:
	UF : 1, UT : 1,
	J1=    90.000 deg,	J2=     0.000 deg
};
P[65]{
   GP1:
	UF : 1, UT : 1,		CONFIG : 'F U T, 0, 0, 0',
	X =  2864.014  mm,	Y =   282.441  mm,	Z =   502.065  mm,
	W =   -15.171 deg,	P =   -43.175 deg,	R =    33.524 deg
   GP2:
	UF : 1, UT : 1,
	J1=    90.000 deg,	J2=     0.000 deg
};
P[66]{
   GP1:
	UF : 1, UT : 1,		CONFIG : 'F U T, 0, 0, 0',
	X =  2896.112  mm,	Y =   278.436  mm,	Z =   463.899  mm,
	W =   -14.926 deg,	P =   -42.904 deg,	R =    33.356 deg
   GP2:
	UF : 1, UT : 1,
	J1=    90.000 deg,	J2=     0.000 deg
};
P[67]{
   GP1:
	UF : 1, UT : 1,		CONFIG : 'F U T, 0, 0, 0',
	X =  2897.490  mm,	Y =   360.733  mm,	Z =   463.056  mm,
	W =    -8.441 deg,	P =   -43.927 deg,	R =    33.763 deg
   GP2:
	UF : 1, UT : 1,
	J1=    90.000 deg,	J2=     0.000 deg
};
P[68]{
   GP1:
	UF : 1, UT : 1,		CONFIG : 'F U T, 0, 0, 0',
	X =  2898.388  mm,	Y =   393.767  mm,	Z =   462.045  mm,
	W =    -2.983 deg,	P =   -44.252 deg,	R =    40.170 deg
   GP2:
	UF : 1, UT : 1,
	J1=    90.000 deg,	J2=     0.000 deg
};
P[69]{
   GP1:
	UF : 1, UT : 1,		CONFIG : 'F U T, 0, 0, 0',
	X =  2895.619  mm,	Y =   404.047  mm,	Z =   461.557  mm,
	W =    -2.617 deg,	P =   -43.939 deg,	R =    53.826 deg
   GP2:
	UF : 1, UT : 1,
	J1=    90.000 deg,	J2=     0.000 deg
};
P[70]{
   GP1:
	UF : 1, UT : 1,		CONFIG : 'F U T, 0, 0, 0',
	X =  2888.819  mm,	Y =   407.185  mm,	Z =   461.271  mm,
	W =    -2.617 deg,	P =   -43.939 deg,	R =    78.094 deg
   GP2:
	UF : 1, UT : 1,
	J1=    90.000 deg,	J2=     0.000 deg
};
P[71]{
   GP1:
	UF : 1, UT : 1,		CONFIG : 'F U T, 0, 0, 0',
	X =  2877.562  mm,	Y =   409.105  mm,	Z =   461.271  mm,
	W =    -2.617 deg,	P =   -43.939 deg,	R =    78.094 deg
   GP2:
	UF : 1, UT : 1,
	J1=    90.000 deg,	J2=     0.000 deg
};
P[72]{
   GP1:
	UF : 1, UT : 1,		CONFIG : 'F U T, 0, 0, 0',
	X =  2697.000  mm,	Y =   247.797  mm,	Z =   648.652  mm,
	W =    -2.629 deg,	P =   -43.936 deg,	R =    42.269 deg
   GP2:
	UF : 1, UT : 1,
	J1=    90.000 deg,	J2=     0.000 deg
};
P[73]{
   GP1:
	UF : 1, UT : 1,		CONFIG : 'N U T, 0, 0, 0',
	X =   949.898  mm,	Y =    98.916  mm,	Z =  1480.357  mm,
	W =   -25.667 deg,	P =   -34.352 deg,	R =    34.753 deg
   GP2:
	UF : 1, UT : 1,
	J1=     0.000 deg,	J2=   180.000 deg
};
P[74]{
   GP1:
	UF : 1, UT : 1,		CONFIG : 'N U T, 1, 0, 0',
	X =  2528.555  mm,	Y =   -65.615  mm,	Z =   892.718  mm,
	W =   -11.578 deg,	P =   -57.733 deg,	R =     8.895 deg
   GP2:
	UF : 1, UT : 1,
	J1=    90.000 deg,	J2=     0.000 deg
};
P[75]{
   GP1:
	UF : 1, UT : 1,		CONFIG : 'N U T, 0, 0, 0',
	X =  2860.056  mm,	Y =  -309.345  mm,	Z =   520.586  mm,
	W =    14.883 deg,	P =   -42.517 deg,	R =   -27.206 deg
   GP2:
	UF : 1, UT : 1,
	J1=    90.000 deg,	J2=     0.000 deg
};
P[76]{
   GP1:
	UF : 1, UT : 1,		CONFIG : 'N U T, 0, 0, 0',
	X =  2897.917  mm,	Y =  -285.431  mm,	Z =   459.923  mm,
	W =    14.883 deg,	P =   -42.517 deg,	R =   -27.206 deg
   GP2:
	UF : 1, UT : 1,
	J1=    90.000 deg,	J2=     0.000 deg
};
P[77]{
   GP1:
	UF : 1, UT : 1,		CONFIG : 'N U T, 0, 0, 0',
	X =  2898.423  mm,	Y =  -384.351  mm,	Z =   461.415  mm,
	W =     7.397 deg,	P =   -43.869 deg,	R =   -27.794 deg
   GP2:
	UF : 1, UT : 1,
	J1=    90.000 deg,	J2=     0.000 deg
};
P[78]{
   GP1:
	UF : 1, UT : 1,		CONFIG : 'N U T, 0, 0, 0',
	X =  2897.209  mm,	Y =  -399.220  mm,	Z =   461.618  mm,
	W =     7.397 deg,	P =   -43.869 deg,	R =   -33.011 deg
   GP2:
	UF : 1, UT : 1,
	J1=    90.000 deg,	J2=     0.000 deg
};
P[79]{
   GP1:
	UF : 1, UT : 1,		CONFIG : 'N U T, 0, 0, 0',
	X =  2894.455  mm,	Y =  -407.278  mm,	Z =   461.615  mm,
	W =    -1.104 deg,	P =   -44.451 deg,	R =   -50.597 deg
   GP2:
	UF : 1, UT : 1,
	J1=    89.997 deg,	J2=     0.000 deg
};
P[80]{
   GP1:
	UF : 1, UT : 1,		CONFIG : 'N U T, 0, 0, 0',
	X =  2890.602  mm,	Y =  -413.663  mm,	Z =   458.117  mm,
	W =    -1.090 deg,	P =   -44.448 deg,	R =   -71.051 deg
   GP2:
	UF : 1, UT : 1,
	J1=    89.995 deg,	J2=     0.000 deg
};
P[81]{
   GP1:
	UF : 1, UT : 1,		CONFIG : 'N U T, 0, 0, 0',
	X =  2876.877  mm,	Y =  -417.188  mm,	Z =   456.595  mm,
	W =    -1.104 deg,	P =   -44.451 deg,	R =   -71.047 deg
   GP2:
	UF : 1, UT : 1,
	J1=    89.995 deg,	J2=     0.000 deg
};
P[82]{
   GP1:
	UF : 1, UT : 1,		CONFIG : 'N U T, 0, 0, 0',
	X =  2690.549  mm,	Y =  -310.856  mm,	Z =   600.282  mm,
	W =     1.613 deg,	P =   -43.868 deg,	R =   -40.404 deg
   GP2:
	UF : 1, UT : 1,
	J1=    90.000 deg,	J2=     0.000 deg
};
P[83]{
   GP1:
	UF : 1, UT : 1,		CONFIG : 'F U T, 0, 0, 0',
	X =  2542.011  mm,	Y =    62.997  mm,	Z =   733.500  mm,
	W =      .337 deg,	P =   -50.731 deg,	R =     6.061 deg
   GP2:
	UF : 1, UT : 1,
	J1=    90.000 deg,	J2=     0.000 deg
};
P[84]{
   GP1:
	UF : 1, UT : 1,		CONFIG : 'F U T, 0, 0, 0',
	X =  2864.014  mm,	Y =   282.441  mm,	Z =   502.065  mm,
	W =   -15.171 deg,	P =   -43.175 deg,	R =    33.524 deg
   GP2:
	UF : 1, UT : 1,
	J1=    90.000 deg,	J2=     0.000 deg
};
P[85]{
   GP1:
	UF : 1, UT : 1,		CONFIG : 'N U T, 0, 0, 0',
	X =  2172.059  mm,	Y =  -149.810  mm,	Z =  -336.475  mm,
	W =    -4.848 deg,	P =     4.640 deg,	R =    10.727 deg
   GP2:
	UF : 1, UT : 1,
	J1=    45.000 deg,	J2=   182.246 deg
};
P[86]{
   GP1:
	UF : 1, UT : 1,		CONFIG : 'N U T, 0, 0, 0',
	X =  1780.474  mm,	Y =    29.584  mm,	Z =   -67.946  mm,
	W =    -4.424 deg,	P =     7.600 deg,	R =    11.037 deg
   GP2:
	UF : 1, UT : 1,
	J1=    45.000 deg,	J2=   182.246 deg
};
P[87]{
   GP1:
	UF : 1, UT : 1,		CONFIG : 'N U T, 0, 0, 0',
	X =  1142.160  mm,	Y =  -217.183  mm,	Z =   141.822  mm,
	W =    36.993 deg,	P =    27.706 deg,	R =  -162.803 deg
   GP2:
	UF : 1, UT : 1,
	J1=    90.000 deg,	J2=   -90.000 deg
};
P[88]{
   GP1:
	UF : 1, UT : 1,		CONFIG : 'N U T, 0, 0, 0',
	X =  1987.244  mm,	Y =     -.972  mm,	Z =  1525.322  mm,
	W =     -.010 deg,	P =    45.000 deg,	R =    90.000 deg
   GP2:
	UF : 1, UT : 1,
	J1=    90.000 deg,	J2=    90.000 deg
};
P[89]{
   GP1:
	UF : 1, UT : 1,		CONFIG : 'N U T, 0, 0, 0',
	X =  2298.943  mm,	Y =    15.028  mm,	Z =   995.580  mm,
	W =   -33.416 deg,	P =    -1.271 deg,	R =    34.407 deg
   GP2:
	UF : 1, UT : 1,
	J1=    89.999 deg,	J2=   -90.000 deg
};
P[90]{
   GP1:
	UF : 1, UT : 1,		CONFIG : 'N U T, 0, 0, -1',
	X =  1457.610  mm,	Y =    -5.074  mm,	Z =    -1.334  mm,
	W =      .944 deg,	P =    42.924 deg,	R =   177.949 deg
   GP2:
	UF : 1, UT : 1,
	J1=     0.000 deg,	J2=   180.000 deg
};
P[91]{
   GP1:
	UF : 1, UT : 1,		CONFIG : 'F U T, 0, 0, 0',
	X =  2701.500  mm,	Y =   248.797  mm,	Z =   650.852  mm,
	W =    -2.629 deg,	P =   -43.936 deg,	R =    42.269 deg
   GP2:
	UF : 1, UT : 1,
	J1=    90.000 deg,	J2=     0.000 deg
};
P[92]{
   GP1:
	UF : 1, UT : 1,		CONFIG : 'F U T, 0, 0, 0',
	X =  2542.011  mm,	Y =    62.997  mm,	Z =   733.500  mm,
	W =      .337 deg,	P =   -50.731 deg,	R =     6.061 deg
   GP2:
	UF : 1, UT : 1,
	J1=    90.000 deg,	J2=     0.000 deg
};
P[93]{
   GP1:
	UF : 1, UT : 1,		CONFIG : 'F U T, 0, 0, 0',
	X =  2864.014  mm,	Y =   282.441  mm,	Z =   502.065  mm,
	W =   -15.171 deg,	P =   -43.175 deg,	R =    33.524 deg
   GP2:
	UF : 1, UT : 1,
	J1=    90.000 deg,	J2=     0.000 deg
};
P[94]{
   GP1:
	UF : 1, UT : 1,		CONFIG : 'N U B, 0, 0, 0',
	X =   356.016  mm,	Y =    -2.054  mm,	Z =  2424.089  mm,
	W =      .020 deg,	P =   -40.008 deg,	R =     -.011 deg
   GP2:
	UF : 1, UT : 1,
	J1=    80.000 deg,	J2=   -90.000 deg
};
P[95]{
   GP1:
	UF : 1, UT : 1,		CONFIG : 'N U T, 0, 0, 1',
	X =  1917.622  mm,	Y =   283.121  mm,	Z =   189.834  mm,
	W =   -26.631 deg,	P =    72.567 deg,	R =   160.596 deg
   GP2:
	UF : 1, UT : 1,
	J1=    80.000 deg,	J2=   -90.000 deg
};
P[96]{
   GP1:
	UF : 1, UT : 1,		CONFIG : 'N U T, 0, 0, 0',
	X =  2368.673  mm,	Y =    45.599  mm,	Z =  1002.320  mm,
	W =     -.010 deg,	P =    44.998 deg,	R =    66.715 deg
   GP2:
	UF : 1, UT : 1,
	J1=    90.000 deg,	J2=    90.000 deg
};
P[97]{
   GP1:
	UF : 1, UT : 1,		CONFIG : 'N U T, 0, 0, 0',
	X =  1913.400  mm,	Y = -1217.274  mm,	Z =  1258.765  mm,
	W =   -40.515 deg,	P =     2.084 deg,	R =   -24.296 deg
   GP2:
	UF : 1, UT : 1,
	J1=   180.000 deg,	J2=   -90.000 deg
};
P[98]{
   GP1:
	UF : 1, UT : 1,		CONFIG : 'N U T, 0, 0, 0',
	X =  1456.823  mm,	Y =  -333.215  mm,	Z =     -.642  mm,
	W =    -1.375 deg,	P =    43.930 deg,	R =   175.836 deg
   GP2:
	UF : 1, UT : 1,
	J1=     0.000 deg,	J2=   180.000 deg
};
P[99]{
   GP1:
	UF : 1, UT : 1,		CONFIG : 'N U T, 0, 0, 0',
	X =  1419.375  mm,	Y =   870.775  mm,	Z =  1903.281  mm,
	W =    32.261 deg,	P =   -18.474 deg,	R =    10.214 deg
   GP2:
	UF : 1, UT : 1,
	J1=   180.000 deg,	J2=    90.000 deg
};
P[100]{
   GP1:
	UF : 1, UT : 1,		CONFIG : 'F U T, 0, 0, 0',
	X =  2701.500  mm,	Y =   248.797  mm,	Z =   650.852  mm,
	W =    -2.629 deg,	P =   -43.936 deg,	R =    42.269 deg
   GP2:
	UF : 1, UT : 1,
	J1=    90.000 deg,	J2=     0.000 deg
};
P[101]{
   GP1:
	UF : 1, UT : 1,		CONFIG : 'N U T, 0, 0, 0',
	X =  1457.144  mm,	Y =  -389.993  mm,	Z =      .340  mm,
	W =     5.164 deg,	P =    43.292 deg,	R =  -179.576 deg
   GP2:
	UF : 1, UT : 1,
	J1=     0.000 deg,	J2=   180.000 deg
};
P[102]{
   GP1:
	UF : 1, UT : 1,		CONFIG : 'N U T, 0, 0, 0',
	X =  2687.056  mm,	Y =  -231.345  mm,	Z =   639.889  mm,
	W =    14.883 deg,	P =   -42.517 deg,	R =   -27.206 deg
   GP2:
	UF : 1, UT : 1,
	J1=    90.000 deg,	J2=     0.000 deg
};
P[103]{
   GP1:
	UF : 1, UT : 1,		CONFIG : 'N U T, 0, 0, 0',
	X =  2860.056  mm,	Y =  -309.345  mm,	Z =   520.586  mm,
	W =    14.883 deg,	P =   -42.517 deg,	R =   -27.206 deg
   GP2:
	UF : 1, UT : 1,
	J1=    90.000 deg,	J2=     0.000 deg
};
P[104]{
   GP1:
	UF : 1, UT : 1,		CONFIG : 'N U B, 0, 0, 0',
	X =   356.007  mm,	Y =    -2.068  mm,	Z =  2424.055  mm,
	W =      .010 deg,	P =   -40.003 deg,	R =     -.004 deg
   GP2:
	UF : 1, UT : 1,
	J1=   180.000 deg,	J2=   150.000 deg
};
P[105]{
   GP1:
	UF : 1, UT : 1,		CONFIG : 'N U T, 0, 0, 0',
	X =  1166.553  mm,	Y = -1374.013  mm,	Z =  1522.225  mm,
	W =   -32.586 deg,	P =   -12.067 deg,	R =    17.529 deg
   GP2:
	UF : 1, UT : 1,
	J1=   180.000 deg,	J2=  -125.000 deg
};
P[106]{
   GP1:
	UF : 1, UT : 1,
	J1=   -55.000 deg,	J2=   -30.678 deg,	J3=    10.000 deg,
	J4=   -84.542 deg,	J5=   -72.333 deg,	J6=   125.863 deg
   GP2:
	UF : 1, UT : 1,
	J1=   100.000 deg,	J2=   -90.000 deg
};
P[107]{
   GP1:
	UF : 1, UT : 1,		CONFIG : 'N U T, 0, 0, 0',
	X =  2337.765  mm,	Y = -1447.908  mm,	Z =  1189.179  mm,
	W =   -45.668 deg,	P =   -29.178 deg,	R =    61.340 deg
   GP2:
	UF : 1, UT : 1,
	J1=   100.000 deg,	J2=   -90.000 deg
};
P[108]{
   GP1:
	UF : 1, UT : 1,		CONFIG : 'N U T, 0, 0, -1',
	X =  2500.465  mm,	Y = -1499.903  mm,	Z =  1059.350  mm,
	W =   -50.284 deg,	P =   -30.325 deg,	R =    67.097 deg
   GP2:
	UF : 0, UT : 1,
	J1=   100.000 deg,	J2=   -90.000 deg
};
P[110]{
   GP1:
	UF : 1, UT : 1,		CONFIG : 'N U T, 0, 0, 0',
	X =  2690.549  mm,	Y =  -310.856  mm,	Z =   600.282  mm,
	W =     1.613 deg,	P =   -43.868 deg,	R =   -40.404 deg
   GP2:
	UF : 1, UT : 1,
	J1=    90.000 deg,	J2=     0.000 deg
};
P[111]{
   GP1:
	UF : 1, UT : 1,		CONFIG : 'N U T, 1, 0, 0',
	X =  2528.555  mm,	Y =   -65.615  mm,	Z =   892.718  mm,
	W =   -11.578 deg,	P =   -57.733 deg,	R =     8.895 deg
   GP2:
	UF : 1, UT : 1,
	J1=    90.000 deg,	J2=     0.000 deg
};
P[112]{
   GP1:
	UF : 1, UT : 1,		CONFIG : 'N U T, 0, 0, 0',
	X =  2860.056  mm,	Y =  -309.345  mm,	Z =   520.586  mm,
	W =    14.883 deg,	P =   -42.517 deg,	R =   -27.206 deg
   GP2:
	UF : 1, UT : 1,
	J1=    90.000 deg,	J2=     0.000 deg
};
P[113]{
   GP1:
	UF : 1, UT : 1,		CONFIG : 'N U T, 0, 0, 0',
	X =  1539.625  mm,	Y = -1470.562  mm,	Z =  1075.975  mm,
	W =   -42.854 deg,	P =   -15.295 deg,	R =    39.123 deg
   GP2:
	UF : 1, UT : 1,
	J1=   180.000 deg,	J2=  -125.000 deg
};
P[114]{
   GP1:
	UF : 1, UT : 1,		CONFIG : 'N U T, 0, 0, 0',
	X =  1851.900  mm,	Y =  1480.079  mm,	Z =  1370.284  mm,
	W =   -15.089 deg,	P =   -28.874 deg,	R =    15.571 deg
   GP2:
	UF : 1, UT : 1,
	J1=    93.119 deg,	J2=    90.000 deg
};
P[115]{
   GP1:
	UF : 1, UT : 1,		CONFIG : 'N U T, 0, 0, 0',
	X =  2526.820  mm,	Y =  1556.392  mm,	Z =  1079.609  mm,
	W =    21.780 deg,	P =   -40.404 deg,	R =   -29.962 deg
   GP2:
	UF : 0, UT : 1,
	J1=    95.000 deg,	J2=    90.000 deg
};
P[116]{
   GP1:
	UF : 1, UT : 1,		CONFIG : 'N U B, 0, 0, 0',
	X =   356.004  mm,	Y =    -2.058  mm,	Z =  2424.066  mm,
	W =      .021 deg,	P =   -40.005 deg,	R =     -.012 deg
   GP2:
	UF : 1, UT : 1,
	J1=   125.000 deg,	J2=     0.000 deg
};
P[117]{
   GP1:
	UF : 1, UT : 1,		CONFIG : 'N U B, 0, 0, 0',
	X =   356.032  mm,	Y =    -2.146  mm,	Z =  2424.050  mm,
	W =      .001 deg,	P =   -40.002 deg,	R =     -.005 deg
   GP2:
	UF : 1, UT : 1,
	J1=     0.000 deg,	J2=   180.000 deg
};
P[118]{
   GP1:
	UF : 1, UT : 1,		CONFIG : 'N U T, 0, 0, 0',
	X =  1214.806  mm,	Y =   169.341  mm,	Z =   386.823  mm,
	W =    23.939 deg,	P =    39.314 deg,	R =  -177.488 deg
   GP2:
	UF : 1, UT : 1,
	J1=    80.000 deg,	J2=   -90.000 deg
};
P[119]{
   GP1:
	UF : 1, UT : 1,		CONFIG : 'N U T, 0, 0, 0',
	X =  2690.549  mm,	Y =  -310.856  mm,	Z =   600.282  mm,
	W =     1.613 deg,	P =   -43.868 deg,	R =   -40.404 deg
   GP2:
	UF : 1, UT : 1,
	J1=    90.000 deg,	J2=     0.000 deg
};
P[120]{
   GP1:
	UF : 1, UT : 1,		CONFIG : 'N U T, 0, 0, 0',
	X =  2420.268  mm,	Y =   -62.420  mm,	Z =   888.262  mm,
	W =     4.742 deg,	P =    44.802 deg,	R =    66.709 deg
   GP2:
	UF : 1, UT : 1,
	J1=    89.999 deg,	J2=    90.000 deg
};
P[121]{
   GP1:
	UF : 1, UT : 1,		CONFIG : 'N U T, 0, 0, -1',
	X =  2671.361  mm,	Y =  -220.509  mm,	Z =   618.788  mm,
	W =    39.952 deg,	P =    49.905 deg,	R =  -159.452 deg
   GP2:
	UF : 1, UT : 1,
	J1=    90.000 deg,	J2=     0.000 deg
};
P[122]{
   GP1:
	UF : 1, UT : 1,		CONFIG : 'N U T, 0, 0, 0',
	X =  2675.436  mm,	Y =  -298.605  mm,	Z =   591.354  mm,
	W =    31.909 deg,	P =    33.590 deg,	R =  -130.034 deg
   GP2:
	UF : 1, UT : 1,
	J1=    90.000 deg,	J2=     0.000 deg
};
P[123]{
   GP1:
	UF : 1, UT : 1,		CONFIG : 'N U T, 0, 0, 0',
	X =  2434.487  mm,	Y =  -113.503  mm,	Z =   886.043  mm,
	W =   -16.311 deg,	P =    44.679 deg,	R =   -47.493 deg
   GP2:
	UF : 1, UT : 1,
	J1=    90.000 deg,	J2=    90.000 deg
};
P[126]{
   GP1:
	UF : 1, UT : 1,		CONFIG : 'N U T, 0, 0, 0',
	X =  2420.624  mm,	Y =  -138.635  mm,	Z =   886.232  mm,
	W =   -16.306 deg,	P =    44.680 deg,	R =   -47.506 deg
   GP2:
	UF : 1, UT : 1,
	J1=    90.000 deg,	J2=    90.000 deg
};
P[127]{
   GP1:
	UF : 1, UT : 1,		CONFIG : 'N U T, 0, 0, 1',
	X =  2781.845  mm,	Y =  -368.449  mm,	Z =   566.925  mm,
	W =    32.749 deg,	P =    20.905 deg,	R =  -102.080 deg
   GP2:
	UF : 1, UT : 1,
	J1=    90.000 deg,	J2=     0.000 deg
};
P[128]{
   GP1:
	UF : 1, UT : 1,		CONFIG : 'N U T, 0, 0, 0',
	X =  2698.335  mm,	Y =   256.194  mm,	Z =   573.763  mm,
	W =   -42.051 deg,	P =    32.739 deg,	R =   124.663 deg
   GP2:
	UF : 1, UT : 1,
	J1=    90.000 deg,	J2=     0.000 deg
};
P[129]{
   GP1:
	UF : 1, UT : 1,		CONFIG : 'N U T, 0, 0, 0',
	X =  2284.980  mm,	Y =  -119.488  mm,	Z =   927.926  mm,
	W =    34.022 deg,	P =    31.444 deg,	R =   -66.610 deg
   GP2:
	UF : 1, UT : 1,
	J1=    90.000 deg,	J2=    90.000 deg
};
P[132]{
   GP1:
	UF : 1, UT : 1,		CONFIG : 'N U T, 0, 0, 0',
	X =  2364.441  mm,	Y =  -140.196  mm,	Z =   874.079  mm,
	W =    33.535 deg,	P =    29.220 deg,	R =   -67.391 deg
   GP2:
	UF : 1, UT : 1,
	J1=    90.000 deg,	J2=    90.000 deg
};
P[133]{
   GP1:
	UF : 1, UT : 1,		CONFIG : 'N U T, 0, 0, 0',
	X =  2750.496  mm,	Y =   369.295  mm,	Z =   531.685  mm,
	W =   -32.204 deg,	P =    27.169 deg,	R =   115.020 deg
   GP2:
	UF : 1, UT : 1,
	J1=    90.000 deg,	J2=     0.000 deg
};
P[134]{
   GP1:
	UF : 1, UT : 1,		CONFIG : 'N U T, 0, 0, 0',
	X =  2433.364  mm,	Y =   -19.547  mm,	Z =   530.114  mm,
	W =    -7.526 deg,	P =    51.572 deg,	R =   125.549 deg
   GP2:
	UF : 1, UT : 1,
	J1=    90.000 deg,	J2=     0.000 deg
};
P[135]{
   GP1:
	UF : 1, UT : 1,		CONFIG : 'N U T, 0, 0, 0',
	X =  1964.092  mm,	Y =   128.072  mm,	Z =   485.282  mm,
	W =    14.025 deg,	P =    31.485 deg,	R =    29.572 deg
   GP2:
	UF : 1, UT : 1,
	J1=    90.000 deg,	J2=     0.000 deg
};
P[136]{
   GP1:
	UF : 1, UT : 1,		CONFIG : 'N U T, 0, 0, 0',
	X =  1776.950  mm,	Y =   181.788  mm,	Z =   449.993  mm,
	W =    35.022 deg,	P =    36.482 deg,	R =    50.220 deg
   GP2:
	UF : 1, UT : 1,
	J1=    90.000 deg,	J2=     0.000 deg
};
P[137]{
   GP1:
	UF : 1, UT : 1,		CONFIG : 'N U T, 0, 0, 0',
	X =  1110.996  mm,	Y =   547.835  mm,	Z =  1204.956  mm,
	W =    30.412 deg,	P =    23.153 deg,	R =   -68.803 deg
   GP2:
	UF : 1, UT : 1,
	J1=    90.000 deg,	J2=    90.000 deg
};
P[138]{
   GP1:
	UF : 1, UT : 1,		CONFIG : 'N U T, 0, 0, 0',
	X =  1746.082  mm,	Y =   249.573  mm,	Z =   569.263  mm,
	W =   -35.537 deg,	P =   -12.977 deg,	R =   -27.038 deg
   GP2:
	UF : 1, UT : 1,
	J1=    90.000 deg,	J2=   100.000 deg
};
P[139]{
   GP1:
	UF : 1, UT : 1,		CONFIG : 'N U T, 0, 0, 0',
	X =  1754.079  mm,	Y =   165.415  mm,	Z =   449.266  mm,
	W =    31.721 deg,	P =    33.769 deg,	R =    48.036 deg
   GP2:
	UF : 1, UT : 1,
	J1=    90.000 deg,	J2=     0.000 deg
};
P[140]{
   GP1:
	UF : 1, UT : 1,		CONFIG : 'N U T, 0, 0, 0',
	X =  1754.079  mm,	Y =  -235.814  mm,	Z =   449.266  mm,
	W =   -34.074 deg,	P =    31.387 deg,	R =   -52.404 deg
   GP2:
	UF : 1, UT : 1,
	J1=    90.000 deg,	J2=     0.000 deg
};
P[141]{
   GP1:
	UF : 1, UT : 1,		CONFIG : 'N U T, 0, 0, 0',
	X =  2157.996  mm,	Y =    56.121  mm,	Z =   156.955  mm,
	W =   -33.684 deg,	P =   -17.646 deg,	R =   -34.041 deg
   GP2:
	UF : 1, UT : 1,
	J1=    90.000 deg,	J2=   100.000 deg
};
P[142]{
   GP1:
	UF : 1, UT : 1,		CONFIG : 'N U T, 0, 0, 0',
	X =  2482.996  mm,	Y =    56.121  mm,	Z =   156.955  mm,
	W =   -33.684 deg,	P =   -17.646 deg,	R =   -34.041 deg
   GP2:
	UF : 1, UT : 1,
	J1=    90.000 deg,	J2=   100.000 deg
};
P[143]{
   GP1:
	UF : 1, UT : 1,		CONFIG : 'N U T, 0, 0, 0',
	X =  1843.198  mm,	Y =  -173.825  mm,	Z =   537.934  mm,
	W =   -34.074 deg,	P =    31.387 deg,	R =   -52.404 deg
   GP2:
	UF : 1, UT : 1,
	J1=    90.000 deg,	J2=     0.000 deg
};
P[144]{
   GP1:
	UF : 1, UT : 1,		CONFIG : 'N U T, 0, 0, 0',
	X =  1807.054  mm,	Y =   -90.826  mm,	Z =  1125.220  mm,
	W =      .036 deg,	P =     1.106 deg,	R =     1.891 deg
   GP2:
	UF : 1, UT : 1,
	J1=    45.000 deg,	J2=     0.000 deg
};
P[145]{
   GP1:
	UF : 1, UT : 1,		CONFIG : 'N U T, 0, 0, 0',
	X =  1807.054  mm,	Y =  -390.825  mm,	Z =  1004.220  mm,
	W =     -.607 deg,	P =      .924 deg,	R =   -33.344 deg
   GP2:
	UF : 1, UT : 1,
	J1=    45.000 deg,	J2=     0.000 deg
};
P[148]{
   GP1:
	UF : 1, UT : 1,		CONFIG : 'N U T, 0, 0, 0',
	X =  1816.054  mm,	Y =  -176.826  mm,	Z =  1084.220  mm,
	W =     -.607 deg,	P =      .924 deg,	R =   -33.344 deg
   GP2:
	UF : 1, UT : 1,
	J1=    45.000 deg,	J2=     0.000 deg
};
P[149]{
   GP1:
	UF : 1, UT : 1,		CONFIG : 'N U T, 0, 0, 0',
	X =  1807.054  mm,	Y =   376.174  mm,	Z =  1018.220  mm,
	W =     -.607 deg,	P =      .924 deg,	R =    40.441 deg
   GP2:
	UF : 1, UT : 1,
	J1=    45.000 deg,	J2=     0.000 deg
};
P[151]{
   GP1:
	UF : 1, UT : 1,		CONFIG : 'N U T, 0, 0, 0',
	X =  2550.156  mm,	Y =    45.835  mm,	Z =   135.483  mm,
	W =   -31.566 deg,	P =   -16.651 deg,	R =   -48.456 deg
   GP2:
	UF : 1, UT : 1,
	J1=    90.000 deg,	J2=   100.000 deg
};
P[152]{
   GP1:
	UF : 1, UT : 1,		CONFIG : 'N U T, 0, 0, 0',
	X =  1807.054  mm,	Y =   173.895  mm,	Z =  1166.219  mm,
	W =     -.607 deg,	P =      .924 deg,	R =    40.441 deg
   GP2:
	UF : 1, UT : 1,
	J1=    45.000 deg,	J2=     0.000 deg
};
P[153]{
   GP1:
	UF : 1, UT : 1,		CONFIG : 'N U T, 0, 0, 0',
	X =   908.243  mm,	Y =     -.972  mm,	Z =  2177.323  mm,
	W =     -.010 deg,	P =   -45.000 deg,	R =     0.000 deg
   GP2:
	UF : 1, UT : 1,
	J1=   125.000 deg,	J2=     0.000 deg
};
P[154]{
   GP1:
	UF : 1, UT : 1,		CONFIG : 'N U T, 0, 0, 0',
	X =  1841.244  mm,	Y =   574.028  mm,	Z =  1589.322  mm,
	W =     -.010 deg,	P =   -11.091 deg,	R =     0.000 deg
   GP2:
	UF : 1, UT : 1,
	J1=   125.000 deg,	J2=     0.000 deg
};
P[155]{
   GP1:
	UF : 1, UT : 1,		CONFIG : 'N U T, 0, 0, 0',
	X =  2130.244  mm,	Y =   574.028  mm,	Z =  1472.322  mm,
	W =     -.010 deg,	P =   -11.091 deg,	R =     0.000 deg
   GP2:
	UF : 1, UT : 1,
	J1=   125.000 deg,	J2=     0.000 deg
};
P[156]{
   GP1:
	UF : 1, UT : 1,		CONFIG : 'N U T, 0, 0, 0',
	X =  2346.710  mm,	Y =    66.661  mm,	Z =   156.955  mm,
	W =   -33.684 deg,	P =   -17.646 deg,	R =   -34.041 deg
   GP2:
	UF : 1, UT : 1,
	J1=    90.000 deg,	J2=   100.000 deg
};
P[159]{
   GP1:
	UF : 1, UT : 1,		CONFIG : 'N U T, 0, 0, 0',
	X =  2192.055  mm,	Y =   448.511  mm,	Z =  1378.272  mm,
	W =     0.000 deg,	P =    -1.567 deg,	R =     0.000 deg
   GP2:
	UF : 1, UT : 1,
	J1=   125.000 deg,	J2=     0.000 deg
};
P[160]{
   GP1:
	UF : 1, UT : 1,		CONFIG : 'N U T, 0, 0, 0',
	X =  2174.054  mm,	Y =    17.763  mm,	Z =  1379.272  mm,
	W =     0.000 deg,	P =    -1.567 deg,	R =     0.000 deg
   GP2:
	UF : 1, UT : 1,
	J1=   125.000 deg,	J2=     0.000 deg
};
P[163]{
   GP1:
	UF : 1, UT : 1,		CONFIG : 'N U T, 0, 0, 0',
	X =  2194.122  mm,	Y =  -401.237  mm,	Z =  1396.402  mm,
	W =     0.000 deg,	P =     1.835 deg,	R =     0.000 deg
   GP2:
	UF : 1, UT : 1,
	J1=   125.000 deg,	J2=     0.000 deg
};
P[164]{
   GP1:
	UF : 1, UT : 1,		CONFIG : 'N U T, 0, 0, 0',
	X =  2176.122  mm,	Y =   354.763  mm,	Z =  1397.402  mm,
	W =     0.000 deg,	P =     1.835 deg,	R =     0.000 deg
   GP2:
	UF : 1, UT : 1,
	J1=   125.000 deg,	J2=     0.000 deg
};
P[167]{
   GP1:
	UF : 1, UT : 1,		CONFIG : 'N U T, 0, 0, 0',
	X =  2176.122  mm,	Y =    15.763  mm,	Z =  1427.402  mm,
	W =     0.000 deg,	P =    -4.591 deg,	R =     0.000 deg
   GP2:
	UF : 1, UT : 1,
	J1=   125.000 deg,	J2=     0.000 deg
};
P[168]{
   GP1:
	UF : 1, UT : 1,		CONFIG : 'N U T, 0, 0, 0',
	X =  2176.122  mm,	Y =  -553.165  mm,	Z =  1427.402  mm,
	W =     0.000 deg,	P =    -4.591 deg,	R =     0.000 deg
   GP2:
	UF : 1, UT : 1,
	J1=   125.000 deg,	J2=     0.000 deg
};
P[172]{
   GP1:
	UF : 1, UT : 1,		CONFIG : 'N U T, 0, 0, 0',
	X =  2174.639  mm,	Y =  -639.399  mm,	Z =  1514.172  mm,
	W =     0.000 deg,	P =   -23.113 deg,	R =     0.000 deg
   GP2:
	UF : 1, UT : 1,
	J1=   125.000 deg,	J2=     0.000 deg
};
P[173]{
   GP1:
	UF : 1, UT : 1,		CONFIG : 'N U T, 0, 0, 0',
	X =  1929.795  mm,	Y =  -639.399  mm,	Z =  1514.172  mm,
	W =     0.000 deg,	P =   -23.113 deg,	R =     0.000 deg
   GP2:
	UF : 1, UT : 1,
	J1=   125.000 deg,	J2=     0.000 deg
};
P[174]{
   GP1:
	UF : 1, UT : 1,		CONFIG : 'N U B, 0, 0, 0',
	X =   356.032  mm,	Y =    -2.146  mm,	Z =  2424.050  mm,
	W =      .001 deg,	P =   -40.002 deg,	R =     -.005 deg
   GP2:
	UF : 1, UT : 1,
	J1=     0.000 deg,	J2=   180.000 deg
};
P[175]{
   GP1:
	UF : 1, UT : 1,		CONFIG : 'N U T, 0, 0, 0',
	X =   908.243  mm,	Y =     -.972  mm,	Z =  1061.322  mm,
	W =     -.010 deg,	P =    45.000 deg,	R =   -90.656 deg
   GP2:
	UF : 1, UT : 1,
	J1=     0.000 deg,	J2=   180.000 deg
};
P[176]{
   GP1:
	UF : 1, UT : 1,		CONFIG : 'N U T, 0, 0, 0',
	X =  2167.744  mm,	Y =   245.457  mm,	Z =   371.894  mm,
	W =    34.980 deg,	P =    30.342 deg,	R =   -11.521 deg
   GP2:
	UF : 1, UT : 1,
	J1=     0.000 deg,	J2=   180.000 deg
};
P[181]{
   GP1:
	UF : 1, UT : 1,		CONFIG : 'N U T, 0, 0, 0',
	X =  2189.474  mm,	Y =   383.790  mm,	Z =   296.220  mm,
